LIN {X 0,Y 258.897,Z 434.556,A -85,B 0,C 180,E1 -20301.928,E2 -20301.928} C_VEL
LIN {X 0,Y 259.548,Z 434.776,A -85,B 0,C 180,E1 -20304.325,E2 -20304.325} C_VEL
LIN {X 0,Y 259.942,Z 436.236,A -85,B 0,C 180,E1 -20306.945,E2 -20306.945} C_VEL
LIN {X 0,Y 259.701,Z 437.624,A -85,B 0,C 180,E1 -20308.285,E2 -20308.285} C_VEL
LIN {X 0,Y 258.705,Z 439.082,A -85,B 0,C 180,E1 -20308.925,E2 -20308.925} C_VEL
LIN {X 0,Y 251.709,Z 446.598,A -85,B 0,C 180,E1 -20311.662,E2 -20311.662} C_VEL
LIN {X 0,Y 246.851,Z 451.078,A -85,B 0,C 180,E1 -20313.813,E2 -20313.813} C_VEL
LIN {X 0,Y 242.381,Z 454.631,A -85,B 0,C 180,E1 -20316.05,E2 -20316.05} C_VEL
LIN {X 0,Y 237.058,Z 458.044,A -85,B 0,C 180,E1 -20319.16,E2 -20319.16} C_VEL
LIN {X 0,Y 232.484,Z 459.981,A -85,B 0,C 180,E1 -20322.404,E2 -20322.404} C_VEL
LIN {X 0,Y 228.635,Z 460.543,A -85,B 0,C 180,E1 -20325.764,E2 -20325.764} C_VEL
LIN {X 0,Y 225.606,Z 459.628,A -85,B 0,C 180,E1 -20329.227,E2 -20329.227} C_VEL
LIN {X 0,Y 223.289,Z 457.297,A -85,B 0,C 180,E1 -20332.767,E2 -20332.767} C_VEL
LIN {X 0,Y 221.729,Z 453.432,A -85,B 0,C 180,E1 -20336.365,E2 -20336.365} C_VEL
LIN {X 0,Y 220.972,Z 447.998,A -85,B 0,C 180,E1 -20340,E2 -20340} C_VEL
LIN {X 0,Y 220.653,Z 441.734,A -85,B 0,C 180,E1 -20343.195,E2 -20343.195} C_VEL
LIN {X 0,Y 220.902,Z 433.929,A -85,B 0,C 180,E1 -20346.393,E2 -20346.393} C_VEL
LIN {X 0,Y 221.552,Z 425.762,A -85,B 0,C 180,E1 -20349.129,E2 -20349.129} C_VEL
LIN {X 0,Y 222.379,Z 415.886,A -85,B 0,C 180,E1 -20351.853,E2 -20351.853} C_VEL
LIN {X 0,Y 223.293,Z 404.919,A -85,B 0,C 180,E1 -20354.351,E2 -20354.351} C_VEL
LIN {X 0,Y 224.497,Z 392.799,A -85,B 0,C 180,E1 -20356.598,E2 -20356.598} C_VEL
LIN {X 0,Y 224.918,Z 385.6,A -85,B 0,C 180,E1 -20357.737,E2 -20357.737} C_VEL
LIN {X 0,Y 221.874,Z 372.126,A -85,B 0,C 180,E1 -20359.633,E2 -20359.633} C_VEL
LIN {X 0,Y 221.004,Z 367.954,A -85,B 0,C 180,E1 -20360.148,E2 -20360.148} C_VEL
LIN {X 0,Y 220.87,Z 367.97,A -85,B 0,C 180,E1 -20364.434,E2 -20364.434} C_VEL
LIN {X 0,Y 220.839,Z 367.975,A -85,B 0,C 180,E1 -20368.513,E2 -20368.513} C_VEL
LIN {X 0,Y 220.826,Z 367.978,A -85,B 0,C 180,E1 -20372.754,E2 -20372.754} C_VEL
LIN {X 0,Y 220.839,Z 367.976,A -85,B 0,C 180,E1 -20377.288,E2 -20377.288} C_VEL
LIN {X 0,Y 220.839,Z 367.975,A -85,B 0,C 180,E1 -20380.201,E2 -20380.201} C_VEL
LIN {X 0,Y 220.805,Z 367.978,A -85,B 0,C 180,E1 -20384.446,E2 -20384.446} C_VEL
LIN {X 0,Y 220.777,Z 367.983,A -85,B 0,C 180,E1 -20388.049,E2 -20388.049} C_VEL
LIN {X 0,Y 220.833,Z 367.977,A -85,B 0,C 180,E1 -20392.794,E2 -20392.794} C_VEL
LIN {X 0,Y 220.825,Z 367.976,A -85,B 0,C 180,E1 -20397.245,E2 -20397.245} C_VEL
LIN {X 0,Y 220.836,Z 367.973,A -85,B 0,C 180,E1 -20401.486,E2 -20401.486} C_VEL
LIN {X 0,Y 220.873,Z 367.97,A -85,B 0,C 180,E1 -20405.566,E2 -20405.566} C_VEL
LIN {X 0,Y 220.91,Z 367.963,A -85,B 0,C 180,E1 -20409.516,E2 -20409.516} C_VEL
LIN {X 0,Y 221.018,Z 367.952,A -85,B 0,C 180,E1 -20413.37,E2 -20413.37} C_VEL
LIN {X 0,Y 221.082,Z 367.943,A -85,B 0,C 180,E1 -20419.004,E2 -20419.004} C_VEL
LIN {X 0,Y 221.26,Z 367.922,A -85,B 0,C 180,E1 -20422.701,E2 -20422.701} C_VEL
LIN {X 0,Y 221.513,Z 367.893,A -85,B 0,C 180,E1 -20428.182,E2 -20428.182} C_VEL
LIN {X 0,Y 221.514,Z 367.893,A -85,B 0,C 180,E1 -20431.818,E2 -20431.818} C_VEL
LIN {X 0,Y 221.26,Z 367.922,A -85,B 0,C 180,E1 -20437.3,E2 -20437.3} C_VEL
LIN {X 0,Y 221.082,Z 367.943,A -85,B 0,C 180,E1 -20440.996,E2 -20440.996} C_VEL
LIN {X 0,Y 221.018,Z 367.952,A -85,B 0,C 180,E1 -20446.63,E2 -20446.63} C_VEL
LIN {X 0,Y 220.894,Z 367.965,A -85,B 0,C 180,E1 -20450.486,E2 -20450.486} C_VEL
LIN {X 0,Y 220.869,Z 367.971,A -85,B 0,C 180,E1 -20454.435,E2 -20454.435} C_VEL
LIN {X 0,Y 220.837,Z 367.973,A -85,B 0,C 180,E1 -20458.514,E2 -20458.514} C_VEL
LIN {X 0,Y 220.826,Z 367.976,A -85,B 0,C 180,E1 -20462.755,E2 -20462.755} C_VEL
LIN {X 0,Y 220.839,Z 367.976,A -85,B 0,C 180,E1 -20467.288,E2 -20467.288} C_VEL
LIN {X 0,Y 220.862,Z 367.972,A -85,B 0,C 180,E1 -20471.932,E2 -20471.932} C_VEL
LIN {X 0,Y 220.792,Z 367.98,A -85,B 0,C 180,E1 -20475.551,E2 -20475.551} C_VEL
LIN {X 0,Y 220.811,Z 367.978,A -85,B 0,C 180,E1 -20480.464,E2 -20480.464} C_VEL
LIN {X 0,Y 220.802,Z 367.979,A -85,B 0,C 180,E1 -20485.046,E2 -20485.046} C_VEL
LIN {X 0,Y 220.87,Z 367.972,A -85,B 0,C 180,E1 -20489.395,E2 -20489.395} C_VEL
LIN {X 0,Y 220.898,Z 367.964,A -85,B 0,C 180,E1 -20493.55,E2 -20493.55} C_VEL
LIN {X 0,Y 220.881,Z 367.97,A -85,B 0,C 180,E1 -20497.554,E2 -20497.554} C_VEL
LIN {X 0,Y 220.988,Z 367.956,A -85,B 0,C 180,E1 -20502.571,E2 -20502.571} C_VEL
LIN {X 0,Y 221.03,Z 367.952,A -85,B 0,C 180,E1 -20507.14,E2 -20507.14} C_VEL
LIN {X 0,Y 221.262,Z 367.921,A -85,B 0,C 180,E1 -20510.862,E2 -20510.862} C_VEL
LIN {X 0,Y 221.315,Z 367.916,A -85,B 0,C 180,E1 -20512.703,E2 -20512.703} C_VEL
LIN {X 0,Y 221.516,Z 367.891,A -85,B 0,C 180,E1 -20518.182,E2 -20518.182} C_VEL
LIN {X 0,Y 221.517,Z 367.889,A -85,B 0,C 180,E1 -20521.818,E2 -20521.818} C_VEL
LIN {X 0,Y 221.258,Z 367.92,A -85,B 0,C 180,E1 -20527.3,E2 -20527.3} C_VEL
LIN {X 0,Y 221.071,Z 367.945,A -85,B 0,C 180,E1 -20530.997,E2 -20530.997} C_VEL
LIN {X 0,Y 221,Z 367.954,A -85,B 0,C 180,E1 -20534.739,E2 -20534.739} C_VEL
LIN {X 0,Y 220.926,Z 367.964,A -85,B 0,C 180,E1 -20538.549,E2 -20538.549} C_VEL
LIN {X 0,Y 220.9,Z 367.967,A -85,B 0,C 180,E1 -20542.683,E2 -20542.683} C_VEL
LIN {X 0,Y 220.887,Z 367.967,A -85,B 0,C 180,E1 -20547.015,E2 -20547.015} C_VEL
LIN {X 0,Y 220.842,Z 367.974,A -85,B 0,C 180,E1 -20550.768,E2 -20550.768} C_VEL
LIN {X 0,Y 220.819,Z 367.974,A -85,B 0,C 180,E1 -20554.952,E2 -20554.952} C_VEL
LIN {X 0,Y 220.984,Z 367.957,A -85,B 0,C 180,E1 -20560.245,E2 -20560.245} C_VEL
LIN {X 0,Y 221.039,Z 368.08,A -85,B 0,C 180,E1 -20560.747,E2 -20560.747} C_VEL
LIN {X 0,Y 222.749,Z 377.209,A -85,B 0,C 180,E1 -20566.526,E2 -20566.526} C_VEL
LIN {X 0,Y 224.08,Z 383.095,A -85,B 0,C 180,E1 -20570.105,E2 -20570.105} C_VEL
LIN {X 0,Y 224.397,Z 385.506,A -85,B 0,C 180,E1 -20571.536,E2 -20571.536} C_VEL
LIN {X 0,Y 223.054,Z 392.251,A -85,B 0,C 180,E1 -20575.448,E2 -20575.448} C_VEL
LIN {X 0,Y 221.469,Z 400.97,A -85,B 0,C 180,E1 -20580.536,E2 -20580.536} C_VEL
LIN {X 0,Y 220.325,Z 410.683,A -85,B 0,C 180,E1 -20586.252,E2 -20586.252} C_VEL
LIN {X 0,Y 220.299,Z 410.997,A -85,B 0,C 180,E1 -20586.436,E2 -20586.436} C_VEL
LIN {X 0,Y 220.113,Z 423.689,A -85,B 0,C 180,E1 -20587.471,E2 -20587.471} C_VEL
LIN {X 0,Y 220.463,Z 437.057,A -85,B 0,C 180,E1 -20588.911,E2 -20588.911} C_VEL
LIN {X 0,Y 220.132,Z 442.349,A -85,B 0,C 180,E1 -20589.594,E2 -20589.594} C_VEL
LIN {X 0,Y 217.709,Z 450.666,A -85,B 0,C 180,E1 -20590.871,E2 -20590.871} C_VEL
LIN {X 0,Y 215.3,Z 458.611,A -85,B 0,C 180,E1 -20592.332,E2 -20592.332} C_VEL
LIN {X 0,Y 214.992,Z 463.305,A -85,B 0,C 180,E1 -20593.279,E2 -20593.279} C_VEL
LIN {X 0,Y 215.345,Z 468.453,A -85,B 0,C 180,E1 -20594.38,E2 -20594.38} C_VEL
LIN {X 0,Y 214.674,Z 477.726,A -85,B 0,C 180,E1 -20596.752,E2 -20596.752} C_VEL
LIN {X 0,Y 214.373,Z 486.701,A -85,B 0,C 180,E1 -20599.585,E2 -20599.585} C_VEL
LIN {X 0,Y 214.461,Z 494.06,A -85,B 0,C 180,E1 -20602.468,E2 -20602.468} C_VEL
LIN {X 0,Y 214.917,Z 499.835,A -85,B 0,C 180,E1 -20605.311,E2 -20605.311} C_VEL
LIN {X 0,Y 215.459,Z 504.208,A -85,B 0,C 180,E1 -20608.131,E2 -20608.131} C_VEL
LIN {X 0,Y 215.668,Z 506.362,A -85,B 0,C 180,E1 -20610,E2 -20610} C_VEL
LIN {X 0,Y 214.924,Z 507.775,A -85,B 0,C 180,E1 -20611.874,E2 -20611.874} C_VEL
LIN {X 0,Y 214.162,Z 508.735,A -85,B 0,C 180,E1 -20613.763,E2 -20613.763} C_VEL
LIN {X 0,Y 213.01,Z 509.516,A -85,B 0,C 180,E1 -20617.584,E2 -20617.584} C_VEL
LIN {X 0,Y 212.759,Z 508.905,A -85,B 0,C 180,E1 -20621.431,E2 -20621.431} C_VEL
LIN {X 0,Y 213.664,Z 507.003,A -85,B 0,C 180,E1 -20625.257,E2 -20625.257} C_VEL
LIN {X 0,Y 215.992,Z 503.521,A -85,B 0,C 180,E1 -20629.332,E2 -20629.332} C_VEL
LIN {X 0,Y 219.285,Z 499.472,A -85,B 0,C 180,E1 -20632.619,E2 -20632.619} C_VEL
LIN {X 0,Y 224.027,Z 493.791,A -85,B 0,C 180,E1 -20636.053,E2 -20636.053} C_VEL
LIN {X 0,Y 229.224,Z 486.787,A -85,B 0,C 180,E1 -20639.377,E2 -20639.377} C_VEL
LIN {X 0,Y 235.31,Z 478.403,A -85,B 0,C 180,E1 -20642.521,E2 -20642.521} C_VEL
LIN {X 0,Y 240.065,Z 470.429,A -85,B 0,C 180,E1 -20645.272,E2 -20645.272} C_VEL
LIN {X 0,Y 244.073,Z 462.536,A -85,B 0,C 180,E1 -20647.96,E2 -20647.96} C_VEL
LIN {X 0,Y 247.623,Z 454.754,A -85,B 0,C 180,E1 -20650.752,E2 -20650.752} C_VEL
LIN {X 0,Y 251.169,Z 447.148,A -85,B 0,C 180,E1 -20653.712,E2 -20653.712} C_VEL
LIN {X 0,Y 252.237,Z 444.781,A -85,B 0,C 180,E1 -20654.827,E2 -20654.827} C_VEL
LIN {X 0,Y 252.529,Z 443.033,A -85,B 0,C 180,E1 -20656.352,E2 -20656.352} C_VEL
LIN {X 0,Y 253.037,Z 441.118,A -85,B 0,C 180,E1 -20658.583,E2 -20658.583} C_VEL
LIN {X 0,Y 253.639,Z 439.942,A -85,B 0,C 180,E1 -20660.882,E2 -20660.882} C_VEL
LIN {X 0,Y 254.229,Z 439.583,A -85,B 0,C 180,E1 -20663.292,E2 -20663.292} C_VEL
LIN {X 0,Y 254.488,Z 439.791,A -85,B 0,C 180,E1 -20664.553,E2 -20664.553} C_VEL
LIN {X 0,Y 254.572,Z 440.686,A -85,B 0,C 180,E1 -20666.485,E2 -20666.485} C_VEL
LIN {X 0,Y 254.481,Z 441.386,A -85,B 0,C 180,E1 -20667.416,E2 -20667.416} C_VEL
LIN {X 0,Y 253.296,Z 442.857,A -85,B 0,C 180,E1 -20668.185,E2 -20668.185} C_VEL
LIN {X 0,Y 246.033,Z 449.795,A -85,B 0,C 180,E1 -20670.947,E2 -20670.947} C_VEL
LIN {X 0,Y 239.373,Z 455.094,A -85,B 0,C 180,E1 -20673.87,E2 -20673.87} C_VEL
LIN {X 0,Y 233.444,Z 458.797,A -85,B 0,C 180,E1 -20676.96,E2 -20676.96} C_VEL
LIN {X 0,Y 228.259,Z 461.111,A -85,B 0,C 180,E1 -20680.203,E2 -20680.203} C_VEL
LIN {X 0,Y 223.761,Z 462.001,A -85,B 0,C 180,E1 -20683.58,E2 -20683.58} C_VEL
LIN {X 0,Y 220.21,Z 461.481,A -85,B 0,C 180,E1 -20687.091,E2 -20687.091} C_VEL
LIN {X 0,Y 217.379,Z 459.554,A -85,B 0,C 180,E1 -20690.697,E2 -20690.697} C_VEL
LIN {X 0,Y 215.348,Z 456.131,A -85,B 0,C 180,E1 -20694.381,E2 -20694.381} C_VEL
LIN {X 0,Y 214.194,Z 451.191,A -85,B 0,C 180,E1 -20698.119,E2 -20698.119} C_VEL
LIN {X 0,Y 213.749,Z 446.372,A -85,B 0,C 180,E1 -20700.942,E2 -20700.942} C_VEL
LIN {X 0,Y 213.555,Z 439.379,A -85,B 0,C 180,E1 -20704.246,E2 -20704.246} C_VEL
LIN {X 0,Y 214.061,Z 430.752,A -85,B 0,C 180,E1 -20707.546,E2 -20707.546} C_VEL
LIN {X 0,Y 214.668,Z 422.303,A -85,B 0,C 180,E1 -20710.194,E2 -20710.194} C_VEL
LIN {X 0,Y 215.588,Z 412.708,A -85,B 0,C 180,E1 -20712.711,E2 -20712.711} C_VEL
LIN {X 0,Y 216.499,Z 402.058,A -85,B 0,C 180,E1 -20715.052,E2 -20715.052} C_VEL
LIN {X 0,Y 217.767,Z 389.029,A -85,B 0,C 180,E1 -20717.369,E2 -20717.369} C_VEL
LIN {X 0,Y 217.714,Z 385.924,A -85,B 0,C 180,E1 -20717.858,E2 -20717.858} C_VEL
LIN {X 0,Y 214.889,Z 373.38,A -85,B 0,C 180,E1 -20719.673,E2 -20719.673} C_VEL
LIN {X 0,Y 213.971,Z 368.83,A -85,B 0,C 180,E1 -20720.299,E2 -20720.299} C_VEL
LIN {X 0,Y 213.804,Z 368.85,A -85,B 0,C 180,E1 -20725.298,E2 -20725.298} C_VEL
LIN {X 0,Y 213.782,Z 368.854,A -85,B 0,C 180,E1 -20729.545,E2 -20729.545} C_VEL
LIN {X 0,Y 213.771,Z 368.852,A -85,B 0,C 180,E1 -20733.979,E2 -20733.979} C_VEL
LIN {X 0,Y 213.78,Z 368.856,A -85,B 0,C 180,E1 -20738.654,E2 -20738.654} C_VEL
LIN {X 0,Y 213.776,Z 368.852,A -85,B 0,C 180,E1 -20743.675,E2 -20743.675} C_VEL
LIN {X 0,Y 213.718,Z 368.863,A -85,B 0,C 180,E1 -20748.876,E2 -20748.876} C_VEL
LIN {X 0,Y 213.754,Z 368.856,A -85,B 0,C 180,E1 -20753.713,E2 -20753.713} C_VEL
LIN {X 0,Y 213.796,Z 368.851,A -85,B 0,C 180,E1 -20758.724,E2 -20758.724} C_VEL
LIN {X 0,Y 213.826,Z 368.851,A -85,B 0,C 180,E1 -20762.603,E2 -20762.603} C_VEL
LIN {X 0,Y 213.863,Z 368.842,A -85,B 0,C 180,E1 -20766.946,E2 -20766.946} C_VEL
LIN {X 0,Y 213.934,Z 368.838,A -85,B 0,C 180,E1 -20772.304,E2 -20772.304} C_VEL
LIN {X 0,Y 213.954,Z 368.829,A -85,B 0,C 180,E1 -20776.707,E2 -20776.707} C_VEL
LIN {X 0,Y 214.143,Z 368.81,A -85,B 0,C 180,E1 -20780.555,E2 -20780.555} C_VEL
LIN {X 0,Y 214.102,Z 368.813,A -85,B 0,C 180,E1 -20784.349,E2 -20784.349} C_VEL
LIN {X 0,Y 214.447,Z 368.774,A -85,B 0,C 180,E1 -20788.122,E2 -20788.122} C_VEL
LIN {X 0,Y 214.551,Z 368.761,A -85,B 0,C 180,E1 -20790,E2 -20790} C_VEL
LIN {X 0,Y 214.447,Z 368.773,A -85,B 0,C 180,E1 -20791.878,E2 -20791.878} C_VEL
LIN {X 0,Y 214.2,Z 368.803,A -85,B 0,C 180,E1 -20797.542,E2 -20797.542} C_VEL
LIN {X 0,Y 214.009,Z 368.825,A -85,B 0,C 180,E1 -20801.364,E2 -20801.364} C_VEL
LIN {X 0,Y 213.935,Z 368.834,A -85,B 0,C 180,E1 -20805.237,E2 -20805.237} C_VEL
LIN {X 0,Y 213.87,Z 368.843,A -85,B 0,C 180,E1 -20809.185,E2 -20809.185} C_VEL
LIN {X 0,Y 213.848,Z 368.845,A -85,B 0,C 180,E1 -20813.227,E2 -20813.227} C_VEL
LIN {X 0,Y 213.83,Z 368.851,A -85,B 0,C 180,E1 -20817.45,E2 -20817.45} C_VEL
LIN {X 0,Y 213.781,Z 368.855,A -85,B 0,C 180,E1 -20821.736,E2 -20821.736} C_VEL
LIN {X 0,Y 213.756,Z 368.856,A -85,B 0,C 180,E1 -20826.286,E2 -20826.286} C_VEL
LIN {X 0,Y 213.799,Z 368.853,A -85,B 0,C 180,E1 -20831.106,E2 -20831.106} C_VEL
LIN {X 0,Y 213.81,Z 368.851,A -85,B 0,C 180,E1 -20833.685,E2 -20833.685} C_VEL
LIN {X 0,Y 213.749,Z 368.855,A -85,B 0,C 180,E1 -20836.333,E2 -20836.333} C_VEL
LIN {X 0,Y 213.727,Z 368.863,A -85,B 0,C 180,E1 -20841.334,E2 -20841.334} C_VEL
LIN {X 0,Y 213.758,Z 368.853,A -85,B 0,C 180,E1 -20846.018,E2 -20846.018} C_VEL
LIN {X 0,Y 213.783,Z 368.854,A -85,B 0,C 180,E1 -20850.455,E2 -20850.455} C_VEL
LIN {X 0,Y 213.805,Z 368.849,A -85,B 0,C 180,E1 -20854.702,E2 -20854.702} C_VEL
LIN {X 0,Y 213.817,Z 368.853,A -85,B 0,C 180,E1 -20858.804,E2 -20858.804} C_VEL
LIN {X 0,Y 213.947,Z 368.833,A -85,B 0,C 180,E1 -20862.804,E2 -20862.804} C_VEL
LIN {X 0,Y 213.985,Z 368.832,A -85,B 0,C 180,E1 -20866.709,E2 -20866.709} C_VEL
LIN {X 0,Y 214.2,Z 368.802,A -85,B 0,C 180,E1 -20870.558,E2 -20870.558} C_VEL
LIN {X 0,Y 214.252,Z 368.794,A -85,B 0,C 180,E1 -20872.461,E2 -20872.461} C_VEL
LIN {X 0,Y 214.45,Z 368.771,A -85,B 0,C 180,E1 -20878.122,E2 -20878.122} C_VEL
LIN {X 0,Y 214.554,Z 368.755,A -85,B 0,C 180,E1 -20880,E2 -20880} C_VEL
LIN {X 0,Y 214.45,Z 368.769,A -85,B 0,C 180,E1 -20881.878,E2 -20881.878} C_VEL
LIN {X 0,Y 214.198,Z 368.8,A -85,B 0,C 180,E1 -20887.542,E2 -20887.542} C_VEL
LIN {X 0,Y 214.003,Z 368.826,A -85,B 0,C 180,E1 -20891.364,E2 -20891.364} C_VEL
LIN {X 0,Y 213.938,Z 368.833,A -85,B 0,C 180,E1 -20895.237,E2 -20895.237} C_VEL
LIN {X 0,Y 213.844,Z 368.845,A -85,B 0,C 180,E1 -20899.187,E2 -20899.187} C_VEL
LIN {X 0,Y 213.851,Z 368.844,A -85,B 0,C 180,E1 -20903.227,E2 -20903.227} C_VEL
LIN {X 0,Y 213.832,Z 368.846,A -85,B 0,C 180,E1 -20907.45,E2 -20907.45} C_VEL
LIN {X 0,Y 213.773,Z 368.857,A -85,B 0,C 180,E1 -20911.737,E2 -20911.737} C_VEL
LIN {X 0,Y 213.76,Z 368.857,A -85,B 0,C 180,E1 -20916.285,E2 -20916.285} C_VEL
LIN {X 0,Y 213.979,Z 368.888,A -85,B 0,C 180,E1 -20920.687,E2 -20920.687} C_VEL
LIN {X 0,Y 215.44,Z 376.781,A -85,B 0,C 180,E1 -20925.863,E2 -20925.863} C_VEL
LIN {X 0,Y 217.06,Z 383.878,A -85,B 0,C 180,E1 -20930.343,E2 -20930.343} C_VEL
LIN {X 0,Y 217.147,Z 386.687,A -85,B 0,C 180,E1 -20932.052,E2 -20932.052} C_VEL
LIN {X 0,Y 215.652,Z 393.822,A -85,B 0,C 180,E1 -20936.356,E2 -20936.356} C_VEL
LIN {X 0,Y 213.908,Z 404.111,A -85,B 0,C 180,E1 -20942.614,E2 -20942.614} C_VEL
LIN {X 0,Y 213.252,Z 410.025,A -85,B 0,C 180,E1 -20946.254,E2 -20946.254} C_VEL
LIN {X 0,Y 213.031,Z 424.1,A -85,B 0,C 180,E1 -20947.48,E2 -20947.48} C_VEL
LIN {X 0,Y 213.397,Z 437.408,A -85,B 0,C 180,E1 -20949.013,E2 -20949.013} C_VEL
LIN {X 0,Y 214.013,Z 449.844,A -85,B 0,C 180,E1 -20950.829,E2 -20950.829} C_VEL
LIN {X 0,Y 214.824,Z 461.312,A -85,B 0,C 180,E1 -20952.876,E2 -20952.876} C_VEL
LIN {X 0,Y 214.992,Z 463.305,A -85,B 0,C 180,E1 -20953.279,E2 -20953.279} C_VEL
LIN {X 0,Y 214.865,Z 466.366,A -85,B 0,C 180,E1 -20953.935,E2 -20953.935} C_VEL
LIN {X 0,Y 213.575,Z 470.619,A -85,B 0,C 180,E1 -20954.981,E2 -20954.981} C_VEL
LIN {X 0,Y 208.863,Z 479.328,A -85,B 0,C 180,E1 -20957.684,E2 -20957.684} C_VEL
LIN {X 0,Y 207.618,Z 482.941,A -85,B 0,C 180,E1 -20958.966,E2 -20958.966} C_VEL
LIN {X 0,Y 207.486,Z 484.164,A -85,B 0,C 180,E1 -20959.405,E2 -20959.405} C_VEL
LIN {X 0,Y 207.583,Z 491.366,A -85,B 0,C 180,E1 -20962.217,E2 -20962.217} C_VEL
LIN {X 0,Y 207.989,Z 497.394,A -85,B 0,C 180,E1 -20965.154,E2 -20965.154} C_VEL
LIN {X 0,Y 208.583,Z 502.045,A -85,B 0,C 180,E1 -20968.069,E2 -20968.069} C_VEL
LIN {X 0,Y 208.814,Z 504.383,A -85,B 0,C 180,E1 -20970,E2 -20970} C_VEL
LIN {X 0,Y 208.039,Z 505.905,A -85,B 0,C 180,E1 -20971.936,E2 -20971.936} C_VEL
LIN {X 0,Y 207.238,Z 506.957,A -85,B 0,C 180,E1 -20973.889,E2 -20973.889} C_VEL
LIN {X 0,Y 206.006,Z 507.927,A -85,B 0,C 180,E1 -20977.843,E2 -20977.843} C_VEL
LIN {X 0,Y 205.809,Z 507.58,A -85,B 0,C 180,E1 -20981.823,E2 -20981.823} C_VEL
LIN {X 0,Y 206.79,Z 505.98,A -85,B 0,C 180,E1 -20985.777,E2 -20985.777} C_VEL
LIN {X 0,Y 209.079,Z 503.076,A -85,B 0,C 180,E1 -20989.745,E2 -20989.745} C_VEL
LIN {X 0,Y 212.729,Z 499.155,A -85,B 0,C 180,E1 -20993.356,E2 -20993.356} C_VEL
LIN {X 0,Y 217.652,Z 493.871,A -85,B 0,C 180,E1 -20996.876,E2 -20996.876} C_VEL
LIN {X 0,Y 223.08,Z 487.324,A -85,B 0,C 180,E1 -21000.27,E2 -21000.27} C_VEL
LIN {X 0,Y 229.425,Z 479.514,A -85,B 0,C 180,E1 -21003.463,E2 -21003.463} C_VEL
LIN {X 0,Y 234.288,Z 472.337,A -85,B 0,C 180,E1 -21006.146,E2 -21006.146} C_VEL
LIN {X 0,Y 238.941,Z 464.382,A -85,B 0,C 180,E1 -21009.084,E2 -21009.084} C_VEL
LIN {X 0,Y 244.322,Z 454.352,A -85,B 0,C 180,E1 -21013.021,E2 -21013.021} C_VEL
LIN {X 0,Y 247.112,Z 449.26,A -85,B 0,C 180,E1 -21015.318,E2 -21015.318} C_VEL
LIN {X 0,Y 247.615,Z 446.997,A -85,B 0,C 180,E1 -21017.558,E2 -21017.558} C_VEL
LIN {X 0,Y 248.211,Z 445.381,A -85,B 0,C 180,E1 -21019.862,E2 -21019.862} C_VEL
LIN {X 0,Y 248.776,Z 444.499,A -85,B 0,C 180,E1 -21022.28,E2 -21022.28} C_VEL
LIN {X 0,Y 249.049,Z 444.399,A -85,B 0,C 180,E1 -21023.657,E2 -21023.657} C_VEL
LIN {X 0,Y 249.121,Z 444.877,A -85,B 0,C 180,E1 -21025.651,E2 -21025.651} C_VEL
LIN {X 0,Y 247.957,Z 446.555,A -85,B 0,C 180,E1 -21027.416,E2 -21027.416} C_VEL
LIN {X 0,Y 240.401,Z 452.958,A -85,B 0,C 180,E1 -21030.199,E2 -21030.199} C_VEL
LIN {X 0,Y 233.444,Z 457.739,A -85,B 0,C 180,E1 -21033.154,E2 -21033.154} C_VEL
LIN {X 0,Y 227.276,Z 461.062,A -85,B 0,C 180,E1 -21036.297,E2 -21036.297} C_VEL
LIN {X 0,Y 221.819,Z 462.953,A -85,B 0,C 180,E1 -21039.603,E2 -21039.603} C_VEL
LIN {X 0,Y 217.117,Z 463.514,A -85,B 0,C 180,E1 -21043.062,E2 -21043.062} C_VEL
LIN {X 0,Y 213.407,Z 462.634,A -85,B 0,C 180,E1 -21046.672,E2 -21046.672} C_VEL
LIN {X 0,Y 210.445,Z 460.353,A -85,B 0,C 180,E1 -21050.387,E2 -21050.387} C_VEL
LIN {X 0,Y 208.302,Z 456.64,A -85,B 0,C 180,E1 -21054.19,E2 -21054.19} C_VEL
LIN {X 0,Y 207.102,Z 451.338,A -85,B 0,C 180,E1 -21058.055,E2 -21058.055} C_VEL
LIN {X 0,Y 206.655,Z 446.258,A -85,B 0,C 180,E1 -21060.974,E2 -21060.974} C_VEL
LIN {X 0,Y 206.487,Z 438.984,A -85,B 0,C 180,E1 -21064.392,E2 -21064.392} C_VEL
LIN {X 0,Y 207.028,Z 429.957,A -85,B 0,C 180,E1 -21067.804,E2 -21067.804} C_VEL
LIN {X 0,Y 207.609,Z 421.66,A -85,B 0,C 180,E1 -21070.401,E2 -21070.401} C_VEL
LIN {X 0,Y 208.63,Z 411.198,A -85,B 0,C 180,E1 -21073.143,E2 -21073.143} C_VEL
LIN {X 0,Y 209.74,Z 398.784,A -85,B 0,C 180,E1 -21075.798,E2 -21075.798} C_VEL
LIN {X 0,Y 210.745,Z 388.038,A -85,B 0,C 180,E1 -21077.681,E2 -21077.681} C_VEL
LIN {X 0,Y 208.156,Z 375.772,A -85,B 0,C 180,E1 -21079.534,E2 -21079.534} C_VEL
LIN {X 0,Y 206.939,Z 369.706,A -85,B 0,C 180,E1 -21080.371,E2 -21080.371} C_VEL
LIN {X 0,Y 206.766,Z 369.726,A -85,B 0,C 180,E1 -21084.072,E2 -21084.072} C_VEL
LIN {X 0,Y 206.746,Z 369.73,A -85,B 0,C 180,E1 -21088.418,E2 -21088.418} C_VEL
LIN {X 0,Y 206.711,Z 369.735,A -85,B 0,C 180,E1 -21092.955,E2 -21092.955} C_VEL
LIN {X 0,Y 206.725,Z 369.733,A -85,B 0,C 180,E1 -21097.73,E2 -21097.73} C_VEL
LIN {X 0,Y 206.694,Z 369.734,A -85,B 0,C 180,E1 -21101.579,E2 -21101.579} C_VEL
LIN {X 0,Y 206.639,Z 369.743,A -85,B 0,C 180,E1 -21105.58,E2 -21105.58} C_VEL
LIN {X 0,Y 206.668,Z 369.738,A -85,B 0,C 180,E1 -21109.75,E2 -21109.75} C_VEL
LIN {X 0,Y 206.732,Z 369.735,A -85,B 0,C 180,E1 -21114.695,E2 -21114.695} C_VEL
LIN {X 0,Y 206.724,Z 369.73,A -85,B 0,C 180,E1 -21119.339,E2 -21119.339} C_VEL
LIN {X 0,Y 206.735,Z 369.732,A -85,B 0,C 180,E1 -21123.772,E2 -21123.772} C_VEL
LIN {X 0,Y 206.779,Z 369.725,A -85,B 0,C 180,E1 -21128.046,E2 -21128.046} C_VEL
LIN {X 0,Y 206.879,Z 369.716,A -85,B 0,C 180,E1 -21132.197,E2 -21132.197} C_VEL
LIN {X 0,Y 206.896,Z 369.711,A -85,B 0,C 180,E1 -21136.244,E2 -21136.244} C_VEL
LIN {X 0,Y 207.1,Z 369.689,A -85,B 0,C 180,E1 -21140.231,E2 -21140.231} C_VEL
LIN {X 0,Y 207.063,Z 369.691,A -85,B 0,C 180,E1 -21144.156,E2 -21144.156} C_VEL
LIN {X 0,Y 207.383,Z 369.653,A -85,B 0,C 180,E1 -21148.058,E2 -21148.058} C_VEL
LIN {X 0,Y 207.516,Z 369.638,A -85,B 0,C 180,E1 -21150,E2 -21150} C_VEL
LIN {X 0,Y 207.384,Z 369.653,A -85,B 0,C 180,E1 -21151.942,E2 -21151.942} C_VEL
LIN {X 0,Y 207.142,Z 369.683,A -85,B 0,C 180,E1 -21157.8,E2 -21157.8} C_VEL
LIN {X 0,Y 206.932,Z 369.707,A -85,B 0,C 180,E1 -21161.758,E2 -21161.758} C_VEL
LIN {X 0,Y 206.869,Z 369.718,A -85,B 0,C 180,E1 -21165.771,E2 -21165.771} C_VEL
LIN {X 0,Y 206.801,Z 369.723,A -85,B 0,C 180,E1 -21169.868,E2 -21169.868} C_VEL
LIN {X 0,Y 206.765,Z 369.729,A -85,B 0,C 180,E1 -21174.072,E2 -21174.072} C_VEL
LIN {X 0,Y 206.745,Z 369.728,A -85,B 0,C 180,E1 -21178.419,E2 -21178.419} C_VEL
LIN {X 0,Y 206.711,Z 369.735,A -85,B 0,C 180,E1 -21182.956,E2 -21182.956} C_VEL
LIN {X 0,Y 206.727,Z 369.73,A -85,B 0,C 180,E1 -21187.73,E2 -21187.73} C_VEL
LIN {X 0,Y 206.727,Z 369.734,A -85,B 0,C 180,E1 -21191.59,E2 -21191.59} C_VEL
LIN {X 0,Y 206.676,Z 369.738,A -85,B 0,C 180,E1 -21195.57,E2 -21195.57} C_VEL
LIN {X 0,Y 206.669,Z 369.74,A -85,B 0,C 180,E1 -21199.751,E2 -21199.751} C_VEL
LIN {X 0,Y 206.701,Z 369.735,A -85,B 0,C 180,E1 -21204.689,E2 -21204.689} C_VEL
LIN {X 0,Y 206.726,Z 369.734,A -85,B 0,C 180,E1 -21209.34,E2 -21209.34} C_VEL
LIN {X 0,Y 206.735,Z 369.728,A -85,B 0,C 180,E1 -21213.773,E2 -21213.773} C_VEL
LIN {X 0,Y 206.761,Z 369.728,A -85,B 0,C 180,E1 -21218.044,E2 -21218.044} C_VEL
LIN {X 0,Y 206.88,Z 369.712,A -85,B 0,C 180,E1 -21222.197,E2 -21222.197} C_VEL
LIN {X 0,Y 206.918,Z 369.709,A -85,B 0,C 180,E1 -21226.246,E2 -21226.246} C_VEL
LIN {X 0,Y 207.137,Z 369.681,A -85,B 0,C 180,E1 -21230.233,E2 -21230.233} C_VEL
LIN {X 0,Y 207.193,Z 369.672,A -85,B 0,C 180,E1 -21232.202,E2 -21232.202} C_VEL
LIN {X 0,Y 207.386,Z 369.651,A -85,B 0,C 180,E1 -21238.058,E2 -21238.058} C_VEL
LIN {X 0,Y 207.519,Z 369.631,A -85,B 0,C 180,E1 -21240,E2 -21240} C_VEL
LIN {X 0,Y 207.386,Z 369.649,A -85,B 0,C 180,E1 -21241.942,E2 -21241.942} C_VEL
LIN {X 0,Y 207.141,Z 369.679,A -85,B 0,C 180,E1 -21247.8,E2 -21247.8} C_VEL
LIN {X 0,Y 206.929,Z 369.708,A -85,B 0,C 180,E1 -21251.758,E2 -21251.758} C_VEL
LIN {X 0,Y 206.872,Z 369.714,A -85,B 0,C 180,E1 -21255.771,E2 -21255.771} C_VEL
LIN {X 0,Y 206.788,Z 369.726,A -85,B 0,C 180,E1 -21259.869,E2 -21259.869} C_VEL
LIN {X 0,Y 206.767,Z 369.728,A -85,B 0,C 180,E1 -21264.072,E2 -21264.072} C_VEL
LIN {X 0,Y 206.74,Z 369.732,A -85,B 0,C 180,E1 -21268.42,E2 -21268.42} C_VEL
LIN {X 0,Y 206.709,Z 369.733,A -85,B 0,C 180,E1 -21272.956,E2 -21272.956} C_VEL
LIN {X 0,Y 206.737,Z 369.733,A -85,B 0,C 180,E1 -21277.728,E2 -21277.728} C_VEL
LIN {X 0,Y 206.942,Z 369.819,A -85,B 0,C 180,E1 -21280.755,E2 -21280.755} C_VEL
LIN {X 0,Y 208.56,Z 378.207,A -85,B 0,C 180,E1 -21286.428,E2 -21286.428} C_VEL
LIN {X 0,Y 210.007,Z 384.49,A -85,B 0,C 180,E1 -21290.517,E2 -21290.517} C_VEL
LIN {X 0,Y 210.076,Z 386.448,A -85,B 0,C 180,E1 -21291.763,E2 -21291.763} C_VEL
LIN {X 0,Y 208.593,Z 393.556,A -85,B 0,C 180,E1 -21296.225,E2 -21296.225} C_VEL
LIN {X 0,Y 206.766,Z 404.081,A -85,B 0,C 180,E1 -21302.885,E2 -21302.885} C_VEL
LIN {X 0,Y 206.235,Z 409.081,A -85,B 0,C 180,E1 -21306.099,E2 -21306.099} C_VEL
LIN {X 0,Y 205.912,Z 422.074,A -85,B 0,C 180,E1 -21307.261,E2 -21307.261} C_VEL
LIN {X 0,Y 206.213,Z 434.967,A -85,B 0,C 180,E1 -21308.77,E2 -21308.77} C_VEL
LIN {X 0,Y 206.871,Z 448.445,A -85,B 0,C 180,E1 -21310.786,E2 -21310.786} C_VEL
LIN {X 0,Y 207.761,Z 460.586,A -85,B 0,C 180,E1 -21313.036,E2 -21313.036} C_VEL
LIN {X 0,Y 208.324,Z 467.686,A -85,B 0,C 180,E1 -21314.593,E2 -21314.593} C_VEL
LIN {X 0,Y 207.679,Z 477.654,A -85,B 0,C 180,E1 -21317.293,E2 -21317.293} C_VEL
LIN {X 0,Y 207.486,Z 484.164,A -85,B 0,C 180,E1 -21319.405,E2 -21319.405} C_VEL
LIN {X 0,Y 206.795,Z 487.552,A -85,B 0,C 180,E1 -21320.733,E2 -21320.733} C_VEL
LIN {X 0,Y 204.234,Z 492.196,A -85,B 0,C 180,E1 -21323.066,E2 -21323.066} C_VEL
LIN {X 0,Y 202.229,Z 495.405,A -85,B 0,C 180,E1 -21325.055,E2 -21325.055} C_VEL
LIN {X 0,Y 201.523,Z 497.722,A -85,B 0,C 180,E1 -21326.605,E2 -21326.605} C_VEL
LIN {X 0,Y 201.539,Z 498.493,A -85,B 0,C 180,E1 -21327.126,E2 -21327.126} C_VEL
LIN {X 0,Y 201.988,Z 502.28,A -85,B 0,C 180,E1 -21330,E2 -21330} C_VEL
LIN {X 0,Y 201.198,Z 503.919,A -85,B 0,C 180,E1 -21332.002,E2 -21332.002} C_VEL
LIN {X 0,Y 200.34,Z 505.097,A -85,B 0,C 180,E1 -21334.023,E2 -21334.023} C_VEL
LIN {X 0,Y 199.046,Z 506.304,A -85,B 0,C 180,E1 -21338.119,E2 -21338.119} C_VEL
LIN {X 0,Y 198.875,Z 506.215,A -85,B 0,C 180,E1 -21342.241,E2 -21342.241} C_VEL
LIN {X 0,Y 199.938,Z 504.896,A -85,B 0,C 180,E1 -21346.332,E2 -21346.332} C_VEL
LIN {X 0,Y 202.315,Z 502.386,A -85,B 0,C 180,E1 -21350.327,E2 -21350.327} C_VEL
LIN {X 0,Y 206.222,Z 498.728,A -85,B 0,C 180,E1 -21354.139,E2 -21354.139} C_VEL
LIN {X 0,Y 211.333,Z 493.864,A -85,B 0,C 180,E1 -21357.748,E2 -21357.748} C_VEL
LIN {X 0,Y 216.988,Z 487.794,A -85,B 0,C 180,E1 -21361.213,E2 -21361.213} C_VEL
LIN {X 0,Y 223.593,Z 480.536,A -85,B 0,C 180,E1 -21364.456,E2 -21364.456} C_VEL
LIN {X 0,Y 228.75,Z 473.772,A -85,B 0,C 180,E1 -21367.202,E2 -21367.202} C_VEL
LIN {X 0,Y 233.824,Z 466.179,A -85,B 0,C 180,E1 -21370.252,E2 -21370.252} C_VEL
LIN {X 0,Y 238.943,Z 457.959,A -85,B 0,C 180,E1 -21373.726,E2 -21373.726} C_VEL
LIN {X 0,Y 241.662,Z 453.735,A -85,B 0,C 180,E1 -21375.735,E2 -21375.735} C_VEL
LIN {X 0,Y 242.409,Z 451.303,A -85,B 0,C 180,E1 -21378.177,E2 -21378.177} C_VEL
LIN {X 0,Y 243.14,Z 449.464,A -85,B 0,C 180,E1 -21381.301,E2 -21381.301} C_VEL
LIN {X 0,Y 243.602,Z 448.978,A -85,B 0,C 180,E1 -21383.883,E2 -21383.883} C_VEL
LIN {X 0,Y 243.62,Z 449.044,A -85,B 0,C 180,E1 -21384.762,E2 -21384.762} C_VEL
LIN {X 0,Y 242.629,Z 450.211,A -85,B 0,C 180,E1 -21386.608,E2 -21386.608} C_VEL
LIN {X 0,Y 234.792,Z 456.026,A -85,B 0,C 180,E1 -21389.412,E2 -21389.412} C_VEL
LIN {X 0,Y 231.064,Z 458.406,A -85,B 0,C 180,E1 -21390.879,E2 -21390.879} C_VEL
LIN {X 0,Y 224.202,Z 461.978,A -85,B 0,C 180,E1 -21393.969,E2 -21393.969} C_VEL
LIN {X 0,Y 218.151,Z 464.173,A -85,B 0,C 180,E1 -21397.257,E2 -21397.257} C_VEL
LIN {X 0,Y 212.855,Z 465.007,A -85,B 0,C 180,E1 -21400.72,E2 -21400.72} C_VEL
LIN {X 0,Y 208.427,Z 464.481,A -85,B 0,C 180,E1 -21404.35,E2 -21404.35} C_VEL
LIN {X 0,Y 204.939,Z 462.588,A -85,B 0,C 180,E1 -21408.126,E2 -21408.126} C_VEL
LIN {X 0,Y 202.297,Z 459.231,A -85,B 0,C 180,E1 -21412.012,E2 -21412.012} C_VEL
LIN {X 0,Y 200.503,Z 454.42,A -85,B 0,C 180,E1 -21415.98,E2 -21415.98} C_VEL
LIN {X 0,Y 199.9,Z 449.727,A -85,B 0,C 180,E1 -21418.992,E2 -21418.992} C_VEL
LIN {X 0,Y 199.413,Z 442.984,A -85,B 0,C 180,E1 -21422.525,E2 -21422.525} C_VEL
LIN {X 0,Y 199.53,Z 434.617,A -85,B 0,C 180,E1 -21426.065,E2 -21426.065} C_VEL
LIN {X 0,Y 200.281,Z 425.977,A -85,B 0,C 180,E1 -21429.085,E2 -21429.085} C_VEL
LIN {X 0,Y 201.111,Z 415.496,A -85,B 0,C 180,E1 -21432.103,E2 -21432.103} C_VEL
LIN {X 0,Y 202.147,Z 403.865,A -85,B 0,C 180,E1 -21434.857,E2 -21434.857} C_VEL
LIN {X 0,Y 203.454,Z 390.92,A -85,B 0,C 180,E1 -21437.333,E2 -21437.333} C_VEL
LIN {X 0,Y 203.595,Z 387.9,A -85,B 0,C 180,E1 -21437.84,E2 -21437.84} C_VEL
LIN {X 0,Y 200.896,Z 375.694,A -85,B 0,C 180,E1 -21439.72,E2 -21439.72} C_VEL
LIN {X 0,Y 199.879,Z 370.585,A -85,B 0,C 180,E1 -21440.443,E2 -21440.443} C_VEL
LIN {X 0,Y 199.675,Z 370.61,A -85,B 0,C 180,E1 -21444.984,E2 -21444.984} C_VEL
LIN {X 0,Y 199.676,Z 370.612,A -85,B 0,C 180,E1 -21449.522,E2 -21449.522} C_VEL
LIN {X 0,Y 199.666,Z 370.612,A -85,B 0,C 180,E1 -21452.352,E2 -21452.352} C_VEL
LIN {X 0,Y 199.654,Z 370.615,A -85,B 0,C 180,E1 -21456.756,E2 -21456.756} C_VEL
LIN {X 0,Y 199.676,Z 370.611,A -85,B 0,C 180,E1 -21459.312,E2 -21459.312} C_VEL
LIN {X 0,Y 199.63,Z 370.615,A -85,B 0,C 180,E1 -21462.327,E2 -21462.327} C_VEL
LIN {X 0,Y 199.598,Z 370.621,A -85,B 0,C 180,E1 -21465.233,E2 -21465.233} C_VEL
LIN {X 0,Y 199.642,Z 370.614,A -85,B 0,C 180,E1 -21470.756,E2 -21470.756} C_VEL
LIN {X 0,Y 199.635,Z 370.616,A -85,B 0,C 180,E1 -21475.718,E2 -21475.718} C_VEL
LIN {X 0,Y 199.705,Z 370.608,A -85,B 0,C 180,E1 -21478.138,E2 -21478.138} C_VEL
LIN {X 0,Y 199.688,Z 370.611,A -85,B 0,C 180,E1 -21482.772,E2 -21482.772} C_VEL
LIN {X 0,Y 199.751,Z 370.599,A -85,B 0,C 180,E1 -21487.231,E2 -21487.231} C_VEL
LIN {X 0,Y 199.838,Z 370.591,A -85,B 0,C 180,E1 -21491.722,E2 -21491.722} C_VEL
LIN {X 0,Y 199.837,Z 370.59,A -85,B 0,C 180,E1 -21495.748,E2 -21495.748} C_VEL
LIN {X 0,Y 200.023,Z 370.568,A -85,B 0,C 180,E1 -21499.882,E2 -21499.882} C_VEL
LIN {X 0,Y 200.025,Z 370.569,A -85,B 0,C 180,E1 -21503.949,E2 -21503.949} C_VEL
LIN {X 0,Y 200.323,Z 370.531,A -85,B 0,C 180,E1 -21507.99,E2 -21507.99} C_VEL
LIN {X 0,Y 200.48,Z 370.514,A -85,B 0,C 180,E1 -21510,E2 -21510} C_VEL
LIN {X 0,Y 200.031,Z 370.565,A -85,B 0,C 180,E1 -21514.03,E2 -21514.03} C_VEL
LIN {X 0,Y 200.09,Z 370.562,A -85,B 0,C 180,E1 -21518.077,E2 -21518.077} C_VEL
LIN {X 0,Y 199.88,Z 370.582,A -85,B 0,C 180,E1 -21522.179,E2 -21522.179} C_VEL
LIN {X 0,Y 199.807,Z 370.595,A -85,B 0,C 180,E1 -21526.344,E2 -21526.344} C_VEL
LIN {X 0,Y 199.825,Z 370.592,A -85,B 0,C 180,E1 -21528.454,E2 -21528.454} C_VEL
LIN {X 0,Y 199.738,Z 370.605,A -85,B 0,C 180,E1 -21533.818,E2 -21533.818} C_VEL
LIN {X 0,Y 199.713,Z 370.604,A -85,B 0,C 180,E1 -21538.387,E2 -21538.387} C_VEL
LIN {X 0,Y 199.665,Z 370.611,A -85,B 0,C 180,E1 -21542.353,E2 -21542.353} C_VEL
LIN {X 0,Y 199.655,Z 370.613,A -85,B 0,C 180,E1 -21546.757,E2 -21546.757} C_VEL
LIN {X 0,Y 199.701,Z 370.606,A -85,B 0,C 180,E1 -21549.307,E2 -21549.307} C_VEL
LIN {X 0,Y 199.665,Z 370.612,A -85,B 0,C 180,E1 -21552.339,E2 -21552.339} C_VEL
LIN {X 0,Y 199.633,Z 370.617,A -85,B 0,C 180,E1 -21555.244,E2 -21555.244} C_VEL
LIN {X 0,Y 199.6,Z 370.618,A -85,B 0,C 180,E1 -21558.011,E2 -21558.011} C_VEL
LIN {X 0,Y 199.616,Z 370.619,A -85,B 0,C 180,E1 -21560.767,E2 -21560.767} C_VEL
LIN {X 0,Y 199.615,Z 370.615,A -85,B 0,C 180,E1 -21565.714,E2 -21565.714} C_VEL
LIN {X 0,Y 199.703,Z 370.607,A -85,B 0,C 180,E1 -21568.138,E2 -21568.138} C_VEL
LIN {X 0,Y 199.69,Z 370.61,A -85,B 0,C 180,E1 -21572.773,E2 -21572.773} C_VEL
LIN {X 0,Y 199.741,Z 370.604,A -85,B 0,C 180,E1 -21577.23,E2 -21577.23} C_VEL
LIN {X 0,Y 199.84,Z 370.588,A -85,B 0,C 180,E1 -21581.722,E2 -21581.722} C_VEL
LIN {X 0,Y 199.852,Z 370.588,A -85,B 0,C 180,E1 -21585.75,E2 -21585.75} C_VEL
LIN {X 0,Y 200.079,Z 370.559,A -85,B 0,C 180,E1 -21589.885,E2 -21589.885} C_VEL
LIN {X 0,Y 200.136,Z 370.55,A -85,B 0,C 180,E1 -21591.926,E2 -21591.926} C_VEL
LIN {X 0,Y 200.326,Z 370.53,A -85,B 0,C 180,E1 -21597.99,E2 -21597.99} C_VEL
LIN {X 0,Y 200.484,Z 370.508,A -85,B 0,C 180,E1 -21600,E2 -21600} C_VEL
LIN {X 0,Y 200.032,Z 370.568,A -85,B 0,C 180,E1 -21604.03,E2 -21604.03} C_VEL
LIN {X 0,Y 200.09,Z 370.559,A -85,B 0,C 180,E1 -21608.077,E2 -21608.077} C_VEL
LIN {X 0,Y 199.879,Z 370.588,A -85,B 0,C 180,E1 -21612.179,E2 -21612.179} C_VEL
LIN {X 0,Y 199.809,Z 370.593,A -85,B 0,C 180,E1 -21616.343,E2 -21616.343} C_VEL
LIN {X 0,Y 199.704,Z 370.608,A -85,B 0,C 180,E1 -21620.605,E2 -21620.605} C_VEL
LIN {X 0,Y 199.677,Z 370.607,A -85,B 0,C 180,E1 -21624.984,E2 -21624.984} C_VEL
LIN {X 0,Y 199.668,Z 370.613,A -85,B 0,C 180,E1 -21629.524,E2 -21629.524} C_VEL
LIN {X 0,Y 199.661,Z 370.612,A -85,B 0,C 180,E1 -21632.35,E2 -21632.35} C_VEL
LIN {X 0,Y 199.661,Z 370.612,A -85,B 0,C 180,E1 -21636.756,E2 -21636.756} C_VEL
LIN {X 0,Y 199.902,Z 370.692,A -85,B 0,C 180,E1 -21640.822,E2 -21640.822} C_VEL
LIN {X 0,Y 201.69,Z 379.567,A -85,B 0,C 180,E1 -21647.034,E2 -21647.034} C_VEL
LIN {X 0,Y 202.927,Z 384.931,A -85,B 0,C 180,E1 -21650.624,E2 -21650.624} C_VEL
LIN {X 0,Y 202.613,Z 388.428,A -85,B 0,C 180,E1 -21652.921,E2 -21652.921} C_VEL
LIN {X 0,Y 200.987,Z 395.649,A -85,B 0,C 180,E1 -21657.651,E2 -21657.651} C_VEL
LIN {X 0,Y 199.728,Z 403.382,A -85,B 0,C 180,E1 -21662.777,E2 -21662.777} C_VEL
LIN {X 0,Y 199.177,Z 408.352,A -85,B 0,C 180,E1 -21665.975,E2 -21665.975} C_VEL
LIN {X 0,Y 198.836,Z 421.946,A -85,B 0,C 180,E1 -21667.257,E2 -21667.257} C_VEL
LIN {X 0,Y 199.124,Z 434.388,A -85,B 0,C 180,E1 -21668.791,E2 -21668.791} C_VEL
LIN {X 0,Y 199.746,Z 446.906,A -85,B 0,C 180,E1 -21670.741,E2 -21670.741} C_VEL
LIN {X 0,Y 200.609,Z 458.49,A -85,B 0,C 180,E1 -21672.938,E2 -21672.938} C_VEL
LIN {X 0,Y 201.329,Z 466.82,A -85,B 0,C 180,E1 -21674.822,E2 -21674.822} C_VEL
LIN {X 0,Y 200.779,Z 475.88,A -85,B 0,C 180,E1 -21677.363,E2 -21677.363} C_VEL
LIN {X 0,Y 200.557,Z 484.745,A -85,B 0,C 180,E1 -21680.418,E2 -21680.418} C_VEL
LIN {X 0,Y 200.843,Z 491.919,A -85,B 0,C 180,E1 -21683.47,E2 -21683.47} C_VEL
LIN {X 0,Y 201.312,Z 496.677,A -85,B 0,C 180,E1 -21685.996,E2 -21685.996} C_VEL
LIN {X 0,Y 201.539,Z 498.493,A -85,B 0,C 180,E1 -21687.126,E2 -21687.126} C_VEL
LIN {X 0,Y 201.323,Z 499.892,A -85,B 0,C 180,E1 -21688.168,E2 -21688.168} C_VEL
LIN {X 0,Y 199.887,Z 501.364,A -85,B 0,C 180,E1 -21689.752,E2 -21689.752} C_VEL
LIN {X 0,Y 196.144,Z 502.745,A -85,B 0,C 180,E1 -21692.433,E2 -21692.433} C_VEL
LIN {X 0,Y 193.076,Z 503.683,A -85,B 0,C 180,E1 -21695.295,E2 -21695.295} C_VEL
LIN {X 0,Y 192.803,Z 503.866,A -85,B 0,C 180,E1 -21695.892,E2 -21695.892} C_VEL
LIN {X 0,Y 192.054,Z 504.638,A -85,B 0,C 180,E1 -21698.869,E2 -21698.869} C_VEL
LIN {X 0,Y 191.993,Z 504.723,A -85,B 0,C 180,E1 -21702.687,E2 -21702.687} C_VEL
LIN {X 0,Y 193.114,Z 503.692,A -85,B 0,C 180,E1 -21706.926,E2 -21706.926} C_VEL
LIN {X 0,Y 195.664,Z 501.519,A -85,B 0,C 180,E1 -21711.05,E2 -21711.05} C_VEL
LIN {X 0,Y 199.743,Z 498.234,A -85,B 0,C 180,E1 -21714.975,E2 -21714.975} C_VEL
LIN {X 0,Y 205.07,Z 493.791,A -85,B 0,C 180,E1 -21718.672,E2 -21718.672} C_VEL
LIN {X 0,Y 210.957,Z 488.185,A -85,B 0,C 180,E1 -21722.211,E2 -21722.211} C_VEL
LIN {X 0,Y 217.818,Z 481.459,A -85,B 0,C 180,E1 -21725.506,E2 -21725.506} C_VEL
LIN {X 0,Y 222.742,Z 475.754,A -85,B 0,C 180,E1 -21728.026,E2 -21728.026} C_VEL
LIN {X 0,Y 227.169,Z 470.024,A -85,B 0,C 180,E1 -21730.518,E2 -21730.518} C_VEL
LIN {X 0,Y 232.711,Z 462.356,A -85,B 0,C 180,E1 -21733.997,E2 -21733.997} C_VEL
LIN {X 0,Y 235.43,Z 458.665,A -85,B 0,C 180,E1 -21735.762,E2 -21735.762} C_VEL
LIN {X 0,Y 236.44,Z 457.002,A -85,B 0,C 180,E1 -21736.869,E2 -21736.869} C_VEL
LIN {X 0,Y 237.337,Z 454.372,A -85,B 0,C 180,E1 -21740.346,E2 -21740.346} C_VEL
LIN {X 0,Y 237.847,Z 453.409,A -85,B 0,C 180,E1 -21742.922,E2 -21742.922} C_VEL
LIN {X 0,Y 237.92,Z 453.277,A -85,B 0,C 180,E1 -21743.787,E2 -21743.787} C_VEL
LIN {X 0,Y 237.193,Z 453.874,A -85,B 0,C 180,E1 -21745.738,E2 -21745.738} C_VEL
LIN {X 0,Y 229.197,Z 459.035,A -85,B 0,C 180,E1 -21748.581,E2 -21748.581} C_VEL
LIN {X 0,Y 221.68,Z 462.914,A -85,B 0,C 180,E1 -21751.604,E2 -21751.604} C_VEL
LIN {X 0,Y 214.944,Z 465.357,A -85,B 0,C 180,E1 -21754.845,E2 -21754.845} C_VEL
LIN {X 0,Y 209.003,Z 466.471,A -85,B 0,C 180,E1 -21758.291,E2 -21758.291} C_VEL
LIN {X 0,Y 203.853,Z 466.292,A -85,B 0,C 180,E1 -21761.923,E2 -21761.923} C_VEL
LIN {X 0,Y 199.787,Z 464.678,A -85,B 0,C 180,E1 -21765.744,E2 -21765.744} C_VEL
LIN {X 0,Y 196.554,Z 461.712,A -85,B 0,C 180,E1 -21769.701,E2 -21769.701} C_VEL
LIN {X 0,Y 194.198,Z 457.309,A -85,B 0,C 180,E1 -21773.767,E2 -21773.767} C_VEL
LIN {X 0,Y 192.93,Z 451.322,A -85,B 0,C 180,E1 -21777.912,E2 -21777.912} C_VEL
LIN {X 0,Y 192.387,Z 444.68,A -85,B 0,C 180,E1 -21781.57,E2 -21781.57} C_VEL
LIN {X 0,Y 192.345,Z 436.428,A -85,B 0,C 180,E1 -21785.241,E2 -21785.241} C_VEL
LIN {X 0,Y 192.982,Z 427.917,A -85,B 0,C 180,E1 -21788.376,E2 -21788.376} C_VEL
LIN {X 0,Y 193.688,Z 418.554,A -85,B 0,C 180,E1 -21791.268,E2 -21791.268} C_VEL
LIN {X 0,Y 194.713,Z 407.424,A -85,B 0,C 180,E1 -21794.101,E2 -21794.101} C_VEL
LIN {X 0,Y 195.924,Z 395.154,A -85,B 0,C 180,E1 -21796.676,E2 -21796.676} C_VEL
LIN {X 0,Y 196.504,Z 389.452,A -85,B 0,C 180,E1 -21797.698,E2 -21797.698} C_VEL
LIN {X 0,Y 193.865,Z 376.689,A -85,B 0,C 180,E1 -21799.737,E2 -21799.737} C_VEL
LIN {X 0,Y 192.846,Z 371.462,A -85,B 0,C 180,E1 -21800.48,E2 -21800.48} C_VEL
LIN {X 0,Y 192.666,Z 371.482,A -85,B 0,C 180,E1 -21804.224,E2 -21804.224} C_VEL
LIN {X 0,Y 192.652,Z 371.488,A -85,B 0,C 180,E1 -21808.892,E2 -21808.892} C_VEL
LIN {X 0,Y 192.602,Z 371.49,A -85,B 0,C 180,E1 -21813.185,E2 -21813.185} C_VEL
LIN {X 0,Y 192.6,Z 371.493,A -85,B 0,C 180,E1 -21818.34,E2 -21818.34} C_VEL
LIN {X 0,Y 192.553,Z 371.497,A -85,B 0,C 180,E1 -21823.115,E2 -21823.115} C_VEL
LIN {X 0,Y 192.52,Z 371.505,A -85,B 0,C 180,E1 -21826.895,E2 -21826.895} C_VEL
LIN {X 0,Y 192.574,Z 371.491,A -85,B 0,C 180,E1 -21831.653,E2 -21831.653} C_VEL
LIN {X 0,Y 192.599,Z 371.493,A -85,B 0,C 180,E1 -21834.278,E2 -21834.278} C_VEL
LIN {X 0,Y 192.608,Z 371.488,A -85,B 0,C 180,E1 -21839.28,E2 -21839.28} C_VEL
LIN {X 0,Y 192.665,Z 371.482,A -85,B 0,C 180,E1 -21841.692,E2 -21841.692} C_VEL
LIN {X 0,Y 192.712,Z 371.48,A -85,B 0,C 180,E1 -21846.349,E2 -21846.349} C_VEL
LIN {X 0,Y 192.782,Z 371.469,A -85,B 0,C 180,E1 -21851.413,E2 -21851.413} C_VEL
LIN {X 0,Y 192.765,Z 371.47,A -85,B 0,C 180,E1 -21855.214,E2 -21855.214} C_VEL
LIN {X 0,Y 192.945,Z 371.449,A -85,B 0,C 180,E1 -21859.567,E2 -21859.567} C_VEL
LIN {X 0,Y 192.987,Z 371.445,A -85,B 0,C 180,E1 -21863.728,E2 -21863.728} C_VEL
LIN {X 0,Y 193.265,Z 371.41,A -85,B 0,C 180,E1 -21867.916,E2 -21867.916} C_VEL
LIN {X 0,Y 193.444,Z 371.39,A -85,B 0,C 180,E1 -21870,E2 -21870} C_VEL
LIN {X 0,Y 192.976,Z 371.443,A -85,B 0,C 180,E1 -21874.177,E2 -21874.177} C_VEL
LIN {X 0,Y 193.037,Z 371.439,A -85,B 0,C 180,E1 -21878.374,E2 -21878.374} C_VEL
LIN {X 0,Y 192.806,Z 371.462,A -85,B 0,C 180,E1 -21882.633,E2 -21882.633} C_VEL
LIN {X 0,Y 192.772,Z 371.471,A -85,B 0,C 180,E1 -21886.958,E2 -21886.958} C_VEL
LIN {X 0,Y 192.644,Z 371.485,A -85,B 0,C 180,E1 -21891.397,E2 -21891.397} C_VEL
LIN {X 0,Y 192.665,Z 371.484,A -85,B 0,C 180,E1 -21894.225,E2 -21894.225} C_VEL
LIN {X 0,Y 192.651,Z 371.484,A -85,B 0,C 180,E1 -21898.893,E2 -21898.893} C_VEL
LIN {X 0,Y 192.601,Z 371.493,A -85,B 0,C 180,E1 -21903.186,E2 -21903.186} C_VEL
LIN {X 0,Y 192.613,Z 371.486,A -85,B 0,C 180,E1 -21908.338,E2 -21908.338} C_VEL
LIN {X 0,Y 192.602,Z 371.495,A -85,B 0,C 180,E1 -21913.131,E2 -21913.131} C_VEL
LIN {X 0,Y 192.539,Z 371.498,A -85,B 0,C 180,E1 -21916.89,E2 -21916.89} C_VEL
LIN {X 0,Y 192.555,Z 371.499,A -85,B 0,C 180,E1 -21921.649,E2 -21921.649} C_VEL
LIN {X 0,Y 192.601,Z 371.49,A -85,B 0,C 180,E1 -21926.815,E2 -21926.815} C_VEL
LIN {X 0,Y 192.667,Z 371.483,A -85,B 0,C 180,E1 -21931.693,E2 -21931.693} C_VEL
LIN {X 0,Y 192.709,Z 371.478,A -85,B 0,C 180,E1 -21936.349,E2 -21936.349} C_VEL
LIN {X 0,Y 192.784,Z 371.467,A -85,B 0,C 180,E1 -21941.414,E2 -21941.414} C_VEL
LIN {X 0,Y 192.857,Z 371.461,A -85,B 0,C 180,E1 -21947.371,E2 -21947.371} C_VEL
LIN {X 0,Y 193.083,Z 371.428,A -85,B 0,C 180,E1 -21951.629,E2 -21951.629} C_VEL
LIN {X 0,Y 193.268,Z 371.409,A -85,B 0,C 180,E1 -21957.916,E2 -21957.916} C_VEL
LIN {X 0,Y 193.447,Z 371.384,A -85,B 0,C 180,E1 -21960,E2 -21960} C_VEL
LIN {X 0,Y 192.978,Z 371.447,A -85,B 0,C 180,E1 -21964.177,E2 -21964.177} C_VEL
LIN {X 0,Y 193.038,Z 371.436,A -85,B 0,C 180,E1 -21968.374,E2 -21968.374} C_VEL
LIN {X 0,Y 192.806,Z 371.468,A -85,B 0,C 180,E1 -21972.633,E2 -21972.633} C_VEL
LIN {X 0,Y 192.762,Z 371.468,A -85,B 0,C 180,E1 -21976.959,E2 -21976.959} C_VEL
LIN {X 0,Y 192.641,Z 371.488,A -85,B 0,C 180,E1 -21981.397,E2 -21981.397} C_VEL
LIN {X 0,Y 192.668,Z 371.483,A -85,B 0,C 180,E1 -21984.225,E2 -21984.225} C_VEL
LIN {X 0,Y 192.647,Z 371.486,A -85,B 0,C 180,E1 -21988.889,E2 -21988.889} C_VEL
LIN {X 0,Y 192.601,Z 371.49,A -85,B 0,C 180,E1 -21993.186,E2 -21993.186} C_VEL
LIN {X 0,Y 192.656,Z 371.486,A -85,B 0,C 180,E1 -21998.328,E2 -21998.328} C_VEL
LIN {X 0,Y 192.906,Z 371.609,A -85,B 0,C 180,E1 -22000.979,E2 -22000.979} C_VEL
LIN {X 0,Y 194.85,Z 381.022,A -85,B 0,C 180,E1 -22007.759,E2 -22007.759} C_VEL
LIN {X 0,Y 195.86,Z 385.794,A -85,B 0,C 180,E1 -22011.086,E2 -22011.086} C_VEL
LIN {X 0,Y 195.23,Z 389.446,A -85,B 0,C 180,E1 -22013.56,E2 -22013.56} C_VEL
LIN {X 0,Y 193.697,Z 396.296,A -85,B 0,C 180,E1 -22018.257,E2 -22018.257} C_VEL
LIN {X 0,Y 192.405,Z 404.538,A -85,B 0,C 180,E1 -22024.003,E2 -22024.003} C_VEL
LIN {X 0,Y 192.154,Z 407.334,A -85,B 0,C 180,E1 -22025.846,E2 -22025.846} C_VEL
LIN {X 0,Y 191.776,Z 420.005,A -85,B 0,C 180,E1 -22027.084,E2 -22027.084} C_VEL
LIN {X 0,Y 192.018,Z 433.511,A -85,B 0,C 180,E1 -22028.811,E2 -22028.811} C_VEL
LIN {X 0,Y 192.712,Z 446.953,A -85,B 0,C 180,E1 -22031.013,E2 -22031.013} C_VEL
LIN {X 0,Y 193.668,Z 458.755,A -85,B 0,C 180,E1 -22033.395,E2 -22033.395} C_VEL
LIN {X 0,Y 194.283,Z 466.814,A -85,B 0,C 180,E1 -22035.332,E2 -22035.332} C_VEL
LIN {X 0,Y 193.79,Z 476.596,A -85,B 0,C 180,E1 -22038.291,E2 -22038.291} C_VEL
LIN {X 0,Y 193.74,Z 484.289,A -85,B 0,C 180,E1 -22041.131,E2 -22041.131} C_VEL
LIN {X 0,Y 194.106,Z 491.25,A -85,B 0,C 180,E1 -22044.285,E2 -22044.285} C_VEL
LIN {X 0,Y 194.756,Z 496.716,A -85,B 0,C 180,E1 -22047.459,E2 -22047.459} C_VEL
LIN {X 0,Y 195.175,Z 500.108,A -85,B 0,C 180,E1 -22050,E2 -22050} C_VEL
LIN {X 0,Y 194.353,Z 501.878,A -85,B 0,C 180,E1 -22052.072,E2 -22052.072} C_VEL
LIN {X 0,Y 192.803,Z 503.866,A -85,B 0,C 180,E1 -22055.892,E2 -22055.892} C_VEL
LIN {X 0,Y 191.685,Z 504.285,A -85,B 0,C 180,E1 -22057.613,E2 -22057.613} C_VEL
LIN {X 0,Y 188.495,Z 504.021,A -85,B 0,C 180,E1 -22060.44,E2 -22060.44} C_VEL
LIN {X 0,Y 186.184,Z 503.437,A -85,B 0,C 180,E1 -22062.765,E2 -22062.765} C_VEL
LIN {X 0,Y 185.446,Z 503.062,A -85,B 0,C 180,E1 -22064.575,E2 -22064.575} C_VEL
LIN {X 0,Y 185.505,Z 502.96,A -85,B 0,C 180,E1 -22065.184,E2 -22065.184} C_VEL
LIN {X 0,Y 187.487,Z 501.644,A -85,B 0,C 180,E1 -22069.717,E2 -22069.717} C_VEL
LIN {X 0,Y 191.046,Z 499.273,A -85,B 0,C 180,E1 -22073.87,E2 -22073.87} C_VEL
LIN {X 0,Y 195.957,Z 495.795,A -85,B 0,C 180,E1 -22077.791,E2 -22077.791} C_VEL
LIN {X 0,Y 201.788,Z 491.194,A -85,B 0,C 180,E1 -22081.496,E2 -22081.496} C_VEL
LIN {X 0,Y 208.498,Z 485.502,A -85,B 0,C 180,E1 -22084.962,E2 -22084.962} C_VEL
LIN {X 0,Y 213.871,Z 480.537,A -85,B 0,C 180,E1 -22087.44,E2 -22087.44} C_VEL
LIN {X 0,Y 220.365,Z 473.462,A -85,B 0,C 180,E1 -22090.829,E2 -22090.829} C_VEL
LIN {X 0,Y 225.614,Z 467.133,A -85,B 0,C 180,E1 -22093.9,E2 -22093.9} C_VEL
LIN {X 0,Y 229.249,Z 462.813,A -85,B 0,C 180,E1 -22096.09,E2 -22096.09} C_VEL
LIN {X 0,Y 230.462,Z 461.234,A -85,B 0,C 180,E1 -22097.045,E2 -22097.045} C_VEL
LIN {X 0,Y 230.917,Z 460.285,A -85,B 0,C 180,E1 -22097.965,E2 -22097.965} C_VEL
LIN {X 0,Y 231.566,Z 458.567,A -85,B 0,C 180,E1 -22100.405,E2 -22100.405} C_VEL
LIN {X 0,Y 232.003,Z 457.565,A -85,B 0,C 180,E1 -22102.709,E2 -22102.709} C_VEL
LIN {X 0,Y 231.585,Z 457.55,A -85,B 0,C 180,E1 -22104.788,E2 -22104.788} C_VEL
LIN {X 0,Y 229.947,Z 458.519,A -85,B 0,C 180,E1 -22105.568,E2 -22105.568} C_VEL
LIN {X 0,Y 223.64,Z 461.987,A -85,B 0,C 180,E1 -22107.708,E2 -22107.708} C_VEL
LIN {X 0,Y 215.815,Z 465.372,A -85,B 0,C 180,E1 -22110.759,E2 -22110.759} C_VEL
LIN {X 0,Y 208.802,Z 467.415,A -85,B 0,C 180,E1 -22114.051,E2 -22114.051} C_VEL
LIN {X 0,Y 202.624,Z 468.11,A -85,B 0,C 180,E1 -22117.571,E2 -22117.571} C_VEL
LIN {X 0,Y 197.242,Z 467.52,A -85,B 0,C 180,E1 -22121.295,E2 -22121.295} C_VEL
LIN {X 0,Y 192.969,Z 465.576,A -85,B 0,C 180,E1 -22125.229,E2 -22125.229} C_VEL
LIN {X 0,Y 189.592,Z 462.236,A -85,B 0,C 180,E1 -22129.318,E2 -22129.318} C_VEL
LIN {X 0,Y 187.144,Z 457.469,A -85,B 0,C 180,E1 -22133.531,E2 -22133.531} C_VEL
LIN {X 0,Y 186.136,Z 452.866,A -85,B 0,C 180,E1 -22136.753,E2 -22136.753} C_VEL
LIN {X 0,Y 185.452,Z 446.293,A -85,B 0,C 180,E1 -22140.542,E2 -22140.542} C_VEL
LIN {X 0,Y 185.273,Z 438.165,A -85,B 0,C 180,E1 -22144.351,E2 -22144.351} C_VEL
LIN {X 0,Y 185.838,Z 428.246,A -85,B 0,C 180,E1 -22148.153,E2 -22148.153} C_VEL
LIN {X 0,Y 186.446,Z 419.733,A -85,B 0,C 180,E1 -22150.863,E2 -22150.863} C_VEL
LIN {X 0,Y 187.549,Z 408.618,A -85,B 0,C 180,E1 -22153.821,E2 -22153.821} C_VEL
LIN {X 0,Y 188.673,Z 396.409,A -85,B 0,C 180,E1 -22156.5,E2 -22156.5} C_VEL
LIN {X 0,Y 189.328,Z 389.188,A -85,B 0,C 180,E1 -22157.833,E2 -22157.833} C_VEL
LIN {X 0,Y 186.502,Z 375.971,A -85,B 0,C 180,E1 -22159.968,E2 -22159.968} C_VEL
LIN {X 0,Y 185.802,Z 372.339,A -85,B 0,C 180,E1 -22160.552,E2 -22160.552} C_VEL
LIN {X 0,Y 185.602,Z 372.363,A -85,B 0,C 180,E1 -22164.662,E2 -22164.662} C_VEL
LIN {X 0,Y 185.58,Z 372.368,A -85,B 0,C 180,E1 -22169.492,E2 -22169.492} C_VEL
LIN {X 0,Y 185.522,Z 372.371,A -85,B 0,C 180,E1 -22174.627,E2 -22174.627} C_VEL
LIN {X 0,Y 185.569,Z 372.369,A -85,B 0,C 180,E1 -22177.313,E2 -22177.313} C_VEL
LIN {X 0,Y 185.523,Z 372.375,A -85,B 0,C 180,E1 -22180.743,E2 -22180.743} C_VEL
LIN {X 0,Y 185.49,Z 372.378,A -85,B 0,C 180,E1 -22186.045,E2 -22186.045} C_VEL
LIN {X 0,Y 185.49,Z 372.376,A -85,B 0,C 180,E1 -22189.901,E2 -22189.901} C_VEL
LIN {X 0,Y 185.544,Z 372.371,A -85,B 0,C 180,E1 -22192.696,E2 -22192.696} C_VEL
LIN {X 0,Y 185.546,Z 372.371,A -85,B 0,C 180,E1 -22197.975,E2 -22197.975} C_VEL
LIN {X 0,Y 185.582,Z 372.365,A -85,B 0,C 180,E1 -22200.576,E2 -22200.576} C_VEL
LIN {X 0,Y 185.606,Z 372.363,A -85,B 0,C 180,E1 -22205.385,E2 -22205.385} C_VEL
LIN {X 0,Y 185.711,Z 372.35,A -85,B 0,C 180,E1 -22211.101,E2 -22211.101} C_VEL
LIN {X 0,Y 185.7,Z 372.352,A -85,B 0,C 180,E1 -22214.638,E2 -22214.638} C_VEL
LIN {X 0,Y 185.889,Z 372.327,A -85,B 0,C 180,E1 -22219.418,E2 -22219.418} C_VEL
LIN {X 0,Y 185.949,Z 372.321,A -85,B 0,C 180,E1 -22223.49,E2 -22223.49} C_VEL
LIN {X 0,Y 186.208,Z 372.288,A -85,B 0,C 180,E1 -22227.837,E2 -22227.837} C_VEL
LIN {X 0,Y 186.408,Z 372.267,A -85,B 0,C 180,E1 -22230,E2 -22230} C_VEL
LIN {X 0,Y 185.923,Z 372.322,A -85,B 0,C 180,E1 -22234.336,E2 -22234.336} C_VEL
LIN {X 0,Y 185.984,Z 372.317,A -85,B 0,C 180,E1 -22238.694,E2 -22238.694} C_VEL
LIN {X 0,Y 185.732,Z 372.343,A -85,B 0,C 180,E1 -22243.123,E2 -22243.123} C_VEL
LIN {X 0,Y 185.718,Z 372.353,A -85,B 0,C 180,E1 -22247.622,E2 -22247.622} C_VEL
LIN {X 0,Y 185.601,Z 372.362,A -85,B 0,C 180,E1 -22252.251,E2 -22252.251} C_VEL
LIN {X 0,Y 185.564,Z 372.37,A -85,B 0,C 180,E1 -22257.032,E2 -22257.032} C_VEL
LIN {X 0,Y 185.58,Z 372.365,A -85,B 0,C 180,E1 -22259.493,E2 -22259.493} C_VEL
LIN {X 0,Y 185.522,Z 372.374,A -85,B 0,C 180,E1 -22264.628,E2 -22264.628} C_VEL
LIN {X 0,Y 185.569,Z 372.367,A -85,B 0,C 180,E1 -22267.314,E2 -22267.314} C_VEL
LIN {X 0,Y 185.573,Z 372.367,A -85,B 0,C 180,E1 -22270.761,E2 -22270.761} C_VEL
LIN {X 0,Y 185.556,Z 372.37,A -85,B 0,C 180,E1 -22273.976,E2 -22273.976} C_VEL
LIN {X 0,Y 185.482,Z 372.38,A -85,B 0,C 180,E1 -22279.272,E2 -22279.272} C_VEL
LIN {X 0,Y 185.509,Z 372.377,A -85,B 0,C 180,E1 -22282.711,E2 -22282.711} C_VEL
LIN {X 0,Y 185.548,Z 372.37,A -85,B 0,C 180,E1 -22287.976,E2 -22287.976} C_VEL
LIN {X 0,Y 185.584,Z 372.368,A -85,B 0,C 180,E1 -22290.576,E2 -22290.576} C_VEL
LIN {X 0,Y 185.59,Z 372.365,A -85,B 0,C 180,E1 -22295.383,E2 -22295.383} C_VEL
LIN {X 0,Y 185.697,Z 372.351,A -85,B 0,C 180,E1 -22301.116,E2 -22301.116} C_VEL
LIN {X 0,Y 185.732,Z 372.348,A -85,B 0,C 180,E1 -22304.641,E2 -22304.641} C_VEL
LIN {X 0,Y 185.946,Z 372.32,A -85,B 0,C 180,E1 -22309.329,E2 -22309.329} C_VEL
LIN {X 0,Y 185.973,Z 372.317,A -85,B 0,C 180,E1 -22313.491,E2 -22313.491} C_VEL
LIN {X 0,Y 186.212,Z 372.288,A -85,B 0,C 180,E1 -22317.837,E2 -22317.837} C_VEL
LIN {X 0,Y 186.411,Z 372.26,A -85,B 0,C 180,E1 -22320,E2 -22320} C_VEL
LIN {X 0,Y 185.924,Z 372.327,A -85,B 0,C 180,E1 -22324.336,E2 -22324.336} C_VEL
LIN {X 0,Y 185.985,Z 372.314,A -85,B 0,C 180,E1 -22328.694,E2 -22328.694} C_VEL
LIN {X 0,Y 185.733,Z 372.348,A -85,B 0,C 180,E1 -22333.123,E2 -22333.123} C_VEL
LIN {X 0,Y 185.694,Z 372.348,A -85,B 0,C 180,E1 -22337.625,E2 -22337.625} C_VEL
LIN {X 0,Y 185.601,Z 372.366,A -85,B 0,C 180,E1 -22342.251,E2 -22342.251} C_VEL
LIN {X 0,Y 185.564,Z 372.366,A -85,B 0,C 180,E1 -22347.032,E2 -22347.032} C_VEL
LIN {X 0,Y 185.581,Z 372.367,A -85,B 0,C 180,E1 -22349.493,E2 -22349.493} C_VEL
LIN {X 0,Y 185.524,Z 372.37,A -85,B 0,C 180,E1 -22354.627,E2 -22354.627} C_VEL
LIN {X 0,Y 185.749,Z 372.347,A -85,B 0,C 180,E1 -22360.032,E2 -22360.032} C_VEL
LIN {X 0,Y 185.845,Z 372.415,A -85,B 0,C 180,E1 -22361.073,E2 -22361.073} C_VEL
LIN {X 0,Y 187.673,Z 381.144,A -85,B 0,C 180,E1 -22367.618,E2 -22367.618} C_VEL
LIN {X 0,Y 188.699,Z 385.407,A -85,B 0,C 180,E1 -22370.716,E2 -22370.716} C_VEL
LIN {X 0,Y 188.535,Z 387.797,A -85,B 0,C 180,E1 -22372.409,E2 -22372.409} C_VEL
LIN {X 0,Y 186.99,Z 394.187,A -85,B 0,C 180,E1 -22376.976,E2 -22376.976} C_VEL
LIN {X 0,Y 185.559,Z 402.439,A -85,B 0,C 180,E1 -22382.967,E2 -22382.967} C_VEL
LIN {X 0,Y 185.156,Z 406.159,A -85,B 0,C 180,E1 -22385.715,E2 -22385.715} C_VEL
LIN {X 0,Y 184.686,Z 418.622,A -85,B 0,C 180,E1 -22386.991,E2 -22386.991} C_VEL
LIN {X 0,Y 184.902,Z 432.436,A -85,B 0,C 180,E1 -22388.833,E2 -22388.833} C_VEL
LIN {X 0,Y 185.641,Z 446.083,A -85,B 0,C 180,E1 -22391.166,E2 -22391.166} C_VEL
LIN {X 0,Y 186.622,Z 457.622,A -85,B 0,C 180,E1 -22393.594,E2 -22393.594} C_VEL
LIN {X 0,Y 187.343,Z 464.681,A -85,B 0,C 180,E1 -22395.332,E2 -22395.332} C_VEL
LIN {X 0,Y 186.941,Z 473.942,A -85,B 0,C 180,E1 -22398.158,E2 -22398.158} C_VEL
LIN {X 0,Y 186.906,Z 482.419,A -85,B 0,C 180,E1 -22401.349,E2 -22401.349} C_VEL
LIN {X 0,Y 187.343,Z 489.474,A -85,B 0,C 180,E1 -22404.618,E2 -22404.618} C_VEL
LIN {X 0,Y 188.026,Z 494.985,A -85,B 0,C 180,E1 -22407.858,E2 -22407.858} C_VEL
LIN {X 0,Y 188.388,Z 497.803,A -85,B 0,C 180,E1 -22410,E2 -22410} C_VEL
LIN {X 0,Y 187.569,Z 499.708,A -85,B 0,C 180,E1 -22412.147,E2 -22412.147} C_VEL
LIN {X 0,Y 185.795,Z 502.093,A -85,B 0,C 180,E1 -22416.516,E2 -22416.516} C_VEL
LIN {X 0,Y 184.998,Z 503.105,A -85,B 0,C 180,E1 -22420.95,E2 -22420.95} C_VEL
LIN {X 0,Y 185.505,Z 502.96,A -85,B 0,C 180,E1 -22425.184,E2 -22425.184} C_VEL
LIN {X 0,Y 185.433,Z 502.581,A -85,B 0,C 180,E1 -22427.007,E2 -22427.007} C_VEL
LIN {X 0,Y 184.125,Z 501.308,A -85,B 0,C 180,E1 -22430.031,E2 -22430.031} C_VEL
LIN {X 0,Y 183.564,Z 499.531,A -85,B 0,C 180,E1 -22433.053,E2 -22433.053} C_VEL
LIN {X 0,Y 184.642,Z 498.365,A -85,B 0,C 180,E1 -22434.815,E2 -22434.815} C_VEL
LIN {X 0,Y 189.714,Z 495.305,A -85,B 0,C 180,E1 -22438.789,E2 -22438.789} C_VEL
LIN {X 0,Y 195.746,Z 491.122,A -85,B 0,C 180,E1 -22442.585,E2 -22442.585} C_VEL
LIN {X 0,Y 202.736,Z 485.91,A -85,B 0,C 180,E1 -22446.109,E2 -22446.109} C_VEL
LIN {X 0,Y 208.28,Z 481.345,A -85,B 0,C 180,E1 -22448.627,E2 -22448.627} C_VEL
LIN {X 0,Y 213.405,Z 476.489,A -85,B 0,C 180,E1 -22451.198,E2 -22451.198} C_VEL
LIN {X 0,Y 218.25,Z 471.483,A -85,B 0,C 180,E1 -22453.815,E2 -22453.815} C_VEL
LIN {X 0,Y 222.901,Z 466.557,A -85,B 0,C 180,E1 -22456.484,E2 -22456.484} C_VEL
LIN {X 0,Y 224.331,Z 465.008,A -85,B 0,C 180,E1 -22457.411,E2 -22457.411} C_VEL
LIN {X 0,Y 225.084,Z 463.801,A -85,B 0,C 180,E1 -22458.537,E2 -22458.537} C_VEL
LIN {X 0,Y 225.792,Z 461.93,A -85,B 0,C 180,E1 -22461.499,E2 -22461.499} C_VEL
LIN {X 0,Y 225.646,Z 461.283,A -85,B 0,C 180,E1 -22464.077,E2 -22464.077} C_VEL
LIN {X 0,Y 222.437,Z 462.867,A -85,B 0,C 180,E1 -22465.339,E2 -22465.339} C_VEL
LIN {X 0,Y 213.955,Z 466.481,A -85,B 0,C 180,E1 -22468.293,E2 -22468.293} C_VEL
LIN {X 0,Y 206.233,Z 468.709,A -85,B 0,C 180,E1 -22471.504,E2 -22471.504} C_VEL
LIN {X 0,Y 199.364,Z 469.659,A -85,B 0,C 180,E1 -22474.974,E2 -22474.974} C_VEL
LIN {X 0,Y 193.321,Z 469.348,A -85,B 0,C 180,E1 -22478.682,E2 -22478.682} C_VEL
LIN {X 0,Y 188.273,Z 467.669,A -85,B 0,C 180,E1 -22482.624,E2 -22482.624} C_VEL
LIN {X 0,Y 184.309,Z 464.656,A -85,B 0,C 180,E1 -22486.774,E2 -22486.774} C_VEL
LIN {X 0,Y 181.257,Z 460.276,A -85,B 0,C 180,E1 -22491.077,E2 -22491.077} C_VEL
LIN {X 0,Y 179.287,Z 454.351,A -85,B 0,C 180,E1 -22495.503,E2 -22495.503} C_VEL
LIN {X 0,Y 178.521,Z 447.832,A -85,B 0,C 180,E1 -22499.436,E2 -22499.436} C_VEL
LIN {X 0,Y 178.153,Z 439.803,A -85,B 0,C 180,E1 -22503.392,E2 -22503.392} C_VEL
LIN {X 0,Y 178.563,Z 430.004,A -85,B 0,C 180,E1 -22507.349,E2 -22507.349} C_VEL
LIN {X 0,Y 179.227,Z 421.655,A -85,B 0,C 180,E1 -22510.163,E2 -22510.163} C_VEL
LIN {X 0,Y 180.337,Z 409.678,A -85,B 0,C 180,E1 -22513.522,E2 -22513.522} C_VEL
LIN {X 0,Y 181.479,Z 397.514,A -85,B 0,C 180,E1 -22516.306,E2 -22516.306} C_VEL
LIN {X 0,Y 182.194,Z 390.383,A -85,B 0,C 180,E1 -22517.684,E2 -22517.684} C_VEL
LIN {X 0,Y 179.808,Z 378.668,A -85,B 0,C 180,E1 -22519.676,E2 -22519.676} C_VEL
LIN {X 0,Y 178.769,Z 373.215,A -85,B 0,C 180,E1 -22520.515,E2 -22520.515} C_VEL
LIN {X 0,Y 178.514,Z 373.243,A -85,B 0,C 180,E1 -22525.662,E2 -22525.662} C_VEL
LIN {X 0,Y 178.502,Z 373.251,A -85,B 0,C 180,E1 -22530.786,E2 -22530.786} C_VEL
LIN {X 0,Y 178.486,Z 373.246,A -85,B 0,C 180,E1 -22534.219,E2 -22534.219} C_VEL
LIN {X 0,Y 178.467,Z 373.255,A -85,B 0,C 180,E1 -22539.055,E2 -22539.055} C_VEL
LIN {X 0,Y 178.439,Z 373.254,A -85,B 0,C 180,E1 -22542.033,E2 -22542.033} C_VEL
LIN {X 0,Y 178.426,Z 373.259,A -85,B 0,C 180,E1 -22545.153,E2 -22545.153} C_VEL
LIN {X 0,Y 178.417,Z 373.261,A -85,B 0,C 180,E1 -22548.454,E2 -22548.454} C_VEL
LIN {X 0,Y 178.45,Z 373.254,A -85,B 0,C 180,E1 -22553.789,E2 -22553.789} C_VEL
LIN {X 0,Y 178.491,Z 373.252,A -85,B 0,C 180,E1 -22556.548,E2 -22556.548} C_VEL
LIN {X 0,Y 178.523,Z 373.243,A -85,B 0,C 180,E1 -22560.006,E2 -22560.006} C_VEL
LIN {X 0,Y 178.535,Z 373.245,A -85,B 0,C 180,E1 -22564.875,E2 -22564.875} C_VEL
LIN {X 0,Y 178.655,Z 373.23,A -85,B 0,C 180,E1 -22570.755,E2 -22570.755} C_VEL
LIN {X 0,Y 178.66,Z 373.226,A -85,B 0,C 180,E1 -22576.348,E2 -22576.348} C_VEL
LIN {X 0,Y 178.912,Z 373.198,A -85,B 0,C 180,E1 -22580.96,E2 -22580.96} C_VEL
LIN {X 0,Y 179.154,Z 373.167,A -85,B 0,C 180,E1 -22587.752,E2 -22587.752} C_VEL
LIN {X 0,Y 179.371,Z 373.143,A -85,B 0,C 180,E1 -22590,E2 -22590} C_VEL
LIN {X 0,Y 178.87,Z 373.199,A -85,B 0,C 180,E1 -22594.507,E2 -22594.507} C_VEL
LIN {X 0,Y 178.912,Z 373.198,A -85,B 0,C 180,E1 -22599.04,E2 -22599.04} C_VEL
LIN {X 0,Y 178.661,Z 373.226,A -85,B 0,C 180,E1 -22603.652,E2 -22603.652} C_VEL
LIN {X 0,Y 178.639,Z 373.232,A -85,B 0,C 180,E1 -22609.231,E2 -22609.231} C_VEL
LIN {X 0,Y 178.535,Z 373.245,A -85,B 0,C 180,E1 -22615.125,E2 -22615.125} C_VEL
LIN {X 0,Y 178.48,Z 373.247,A -85,B 0,C 180,E1 -22620.791,E2 -22620.791} C_VEL
LIN {X 0,Y 178.486,Z 373.251,A -85,B 0,C 180,E1 -22624.22,E2 -22624.22} C_VEL
LIN {X 0,Y 178.482,Z 373.248,A -85,B 0,C 180,E1 -22629.053,E2 -22629.053} C_VEL
LIN {X 0,Y 178.502,Z 373.249,A -85,B 0,C 180,E1 -22632.016,E2 -22632.016} C_VEL
LIN {X 0,Y 178.458,Z 373.255,A -85,B 0,C 180,E1 -22635.144,E2 -22635.144} C_VEL
LIN {X 0,Y 178.419,Z 373.256,A -85,B 0,C 180,E1 -22638.454,E2 -22638.454} C_VEL
LIN {X 0,Y 178.425,Z 373.256,A -85,B 0,C 180,E1 -22643.784,E2 -22643.784} C_VEL
LIN {X 0,Y 178.489,Z 373.247,A -85,B 0,C 180,E1 -22646.548,E2 -22646.548} C_VEL
LIN {X 0,Y 178.525,Z 373.246,A -85,B 0,C 180,E1 -22650.007,E2 -22650.007} C_VEL
LIN {X 0,Y 178.537,Z 373.242,A -85,B 0,C 180,E1 -22654.876,E2 -22654.876} C_VEL
LIN {X 0,Y 178.641,Z 373.232,A -85,B 0,C 180,E1 -22660.77,E2 -22660.77} C_VEL
LIN {X 0,Y 178.679,Z 373.224,A -85,B 0,C 180,E1 -22664.019,E2 -22664.019} C_VEL
LIN {X 0,Y 178.898,Z 373.198,A -85,B 0,C 180,E1 -22669.154,E2 -22669.154} C_VEL
LIN {X 0,Y 178.938,Z 373.194,A -85,B 0,C 180,E1 -22673.234,E2 -22673.234} C_VEL
LIN {X 0,Y 179.158,Z 373.166,A -85,B 0,C 180,E1 -22677.752,E2 -22677.752} C_VEL
LIN {X 0,Y 179.374,Z 373.137,A -85,B 0,C 180,E1 -22680,E2 -22680} C_VEL
LIN {X 0,Y 178.871,Z 373.205,A -85,B 0,C 180,E1 -22684.507,E2 -22684.507} C_VEL
LIN {X 0,Y 178.914,Z 373.194,A -85,B 0,C 180,E1 -22689.041,E2 -22689.041} C_VEL
LIN {X 0,Y 178.662,Z 373.229,A -85,B 0,C 180,E1 -22693.652,E2 -22693.652} C_VEL
LIN {X 0,Y 178.627,Z 373.232,A -85,B 0,C 180,E1 -22699.217,E2 -22699.217} C_VEL
LIN {X 0,Y 178.538,Z 373.24,A -85,B 0,C 180,E1 -22705.124,E2 -22705.124} C_VEL
LIN {X 0,Y 178.48,Z 373.251,A -85,B 0,C 180,E1 -22710.791,E2 -22710.791} C_VEL
LIN {X 0,Y 178.487,Z 373.248,A -85,B 0,C 180,E1 -22714.219,E2 -22714.219} C_VEL
LIN {X 0,Y 178.728,Z 373.22,A -85,B 0,C 180,E1 -22720.376,E2 -22720.376} C_VEL
LIN {X 0,Y 178.855,Z 373.305,A -85,B 0,C 180,E1 -22721.302,E2 -22721.302} C_VEL
LIN {X 0,Y 180.576,Z 381.497,A -85,B 0,C 180,E1 -22727.687,E2 -22727.687} C_VEL
LIN {X 0,Y 181.574,Z 385.525,A -85,B 0,C 180,E1 -22730.726,E2 -22730.726} C_VEL
LIN {X 0,Y 181.158,Z 388.629,A -85,B 0,C 180,E1 -22733.035,E2 -22733.035} C_VEL
LIN {X 0,Y 179.555,Z 395.371,A -85,B 0,C 180,E1 -22738.102,E2 -22738.102} C_VEL
LIN {X 0,Y 178.26,Z 403.446,A -85,B 0,C 180,E1 -22744.298,E2 -22744.298} C_VEL
LIN {X 0,Y 178.134,Z 405.184,A -85,B 0,C 180,E1 -22745.624,E2 -22745.624} C_VEL
LIN {X 0,Y 177.604,Z 417.882,A -85,B 0,C 180,E1 -22746.997,E2 -22746.997} C_VEL
LIN {X 0,Y 177.813,Z 431.198,A -85,B 0,C 180,E1 -22748.859,E2 -22748.859} C_VEL
LIN {X 0,Y 178.552,Z 444.057,A -85,B 0,C 180,E1 -22751.133,E2 -22751.133} C_VEL
LIN {X 0,Y 179.595,Z 456.376,A -85,B 0,C 180,E1 -22753.81,E2 -22753.81} C_VEL
LIN {X 0,Y 180.392,Z 464.469,A -85,B 0,C 180,E1 -22755.907,E2 -22755.907} C_VEL
LIN {X 0,Y 180.071,Z 474.789,A -85,B 0,C 180,E1 -22759.316,E2 -22759.316} C_VEL
LIN {X 0,Y 180.21,Z 483.055,A -85,B 0,C 180,E1 -22762.718,E2 -22762.718} C_VEL
LIN {X 0,Y 180.666,Z 488.653,A -85,B 0,C 180,E1 -22765.538,E2 -22765.538} C_VEL
LIN {X 0,Y 181.406,Z 493.983,A -85,B 0,C 180,E1 -22768.89,E2 -22768.89} C_VEL
LIN {X 0,Y 181.597,Z 495.404,A -85,B 0,C 180,E1 -22770,E2 -22770} C_VEL
LIN {X 0,Y 180.796,Z 497.467,A -85,B 0,C 180,E1 -22772.228,E2 -22772.228} C_VEL
LIN {X 0,Y 178.927,Z 500.071,A -85,B 0,C 180,E1 -22776.767,E2 -22776.767} C_VEL
LIN {X 0,Y 178.135,Z 501.313,A -85,B 0,C 180,E1 -22781.377,E2 -22781.377} C_VEL
LIN {X 0,Y 178.754,Z 501.411,A -85,B 0,C 180,E1 -22785.975,E2 -22785.975} C_VEL
LIN {X 0,Y 180.842,Z 500.427,A -85,B 0,C 180,E1 -22790.473,E2 -22790.473} C_VEL
LIN {X 0,Y 184.642,Z 498.365,A -85,B 0,C 180,E1 -22794.815,E2 -22794.815} C_VEL
LIN {X 0,Y 185.957,Z 497.184,A -85,B 0,C 180,E1 -22796.557,E2 -22796.557} C_VEL
LIN {X 0,Y 186.818,Z 494.875,A -85,B 0,C 180,E1 -22799.517,E2 -22799.517} C_VEL
LIN {X 0,Y 187.76,Z 492.852,A -85,B 0,C 180,E1 -22801.85,E2 -22801.85} C_VEL
LIN {X 0,Y 189.428,Z 491.205,A -85,B 0,C 180,E1 -22803.498,E2 -22803.498} C_VEL
LIN {X 0,Y 190.263,Z 490.624,A -85,B 0,C 180,E1 -22804.008,E2 -22804.008} C_VEL
LIN {X 0,Y 199.029,Z 484.843,A -85,B 0,C 180,E1 -22808.167,E2 -22808.167} C_VEL
LIN {X 0,Y 205.56,Z 479.73,A -85,B 0,C 180,E1 -22811.221,E2 -22811.221} C_VEL
LIN {X 0,Y 211.518,Z 474.442,A -85,B 0,C 180,E1 -22814.248,E2 -22814.248} C_VEL
LIN {X 0,Y 216.668,Z 469.63,A -85,B 0,C 180,E1 -22817.064,E2 -22817.064} C_VEL
LIN {X 0,Y 218.004,Z 468.382,A -85,B 0,C 180,E1 -22817.857,E2 -22817.857} C_VEL
LIN {X 0,Y 218.979,Z 467.209,A -85,B 0,C 180,E1 -22818.881,E2 -22818.881} C_VEL
LIN {X 0,Y 219.304,Z 466.26,A -85,B 0,C 180,E1 -22820.276,E2 -22820.276} C_VEL
LIN {X 0,Y 219.53,Z 464.955,A -85,B 0,C 180,E1 -22823.164,E2 -22823.164} C_VEL
LIN {X 0,Y 217.074,Z 465.877,A -85,B 0,C 180,E1 -22824.354,E2 -22824.354} C_VEL
LIN {X 0,Y 208.307,Z 468.981,A -85,B 0,C 180,E1 -22827.328,E2 -22827.328} C_VEL
LIN {X 0,Y 200.295,Z 470.792,A -85,B 0,C 180,E1 -22830.578,E2 -22830.578} C_VEL
LIN {X 0,Y 193.135,Z 471.299,A -85,B 0,C 180,E1 -22834.108,E2 -22834.108} C_VEL
LIN {X 0,Y 186.833,Z 470.565,A -85,B 0,C 180,E1 -22837.903,E2 -22837.903} C_VEL
LIN {X 0,Y 181.56,Z 468.531,A -85,B 0,C 180,E1 -22841.96,E2 -22841.96} C_VEL
LIN {X 0,Y 177.42,Z 465.122,A -85,B 0,C 180,E1 -22846.25,E2 -22846.25} C_VEL
LIN {X 0,Y 174.247,Z 460.35,A -85,B 0,C 180,E1 -22850.715,E2 -22850.715} C_VEL
LIN {X 0,Y 172.226,Z 454.075,A -85,B 0,C 180,E1 -22855.318,E2 -22855.318} C_VEL
LIN {X 0,Y 171.373,Z 446.092,A -85,B 0,C 180,E1 -22860,E2 -22860} C_VEL
LIN {X 0,Y 171.128,Z 437.426,A -85,B 0,C 180,E1 -22864.121,E2 -22864.121} C_VEL
LIN {X 0,Y 171.726,Z 426.902,A -85,B 0,C 180,E1 -22868.235,E2 -22868.235} C_VEL
LIN {X 0,Y 172.583,Z 415.85,A -85,B 0,C 180,E1 -22871.748,E2 -22871.748} C_VEL
LIN {X 0,Y 173.624,Z 404.823,A -85,B 0,C 180,E1 -22874.654,E2 -22874.654} C_VEL
LIN {X 0,Y 174.839,Z 392.872,A -85,B 0,C 180,E1 -22877.244,E2 -22877.244} C_VEL
LIN {X 0,Y 175.002,Z 389.831,A -85,B 0,C 180,E1 -22877.831,E2 -22877.831} C_VEL
LIN {X 0,Y 172.141,Z 376.334,A -85,B 0,C 180,E1 -22880.111,E2 -22880.111} C_VEL
LIN {X 0,Y 171.752,Z 374.089,A -85,B 0,C 180,E1 -22880.465,E2 -22880.465} C_VEL
LIN {X 0,Y 171.42,Z 374.128,A -85,B 0,C 180,E1 -22886.807,E2 -22886.807} C_VEL
LIN {X 0,Y 171.459,Z 374.127,A -85,B 0,C 180,E1 -22890.596,E2 -22890.596} C_VEL
LIN {X 0,Y 171.405,Z 374.13,A -85,B 0,C 180,E1 -22895.031,E2 -22895.031} C_VEL
LIN {X 0,Y 171.422,Z 374.133,A -85,B 0,C 180,E1 -22898.834,E2 -22898.834} C_VEL
LIN {X 0,Y 171.352,Z 374.136,A -85,B 0,C 180,E1 -22904.207,E2 -22904.207} C_VEL
LIN {X 0,Y 171.349,Z 374.139,A -85,B 0,C 180,E1 -22908.985,E2 -22908.985} C_VEL
LIN {X 0,Y 171.414,Z 374.127,A -85,B 0,C 180,E1 -22912.048,E2 -22912.048} C_VEL
LIN {X 0,Y 171.411,Z 374.133,A -85,B 0,C 180,E1 -22915.086,E2 -22915.086} C_VEL
LIN {X 0,Y 171.45,Z 374.125,A -85,B 0,C 180,E1 -22920.534,E2 -22920.534} C_VEL
LIN {X 0,Y 171.466,Z 374.125,A -85,B 0,C 180,E1 -22925.803,E2 -22925.803} C_VEL
LIN {X 0,Y 171.611,Z 374.107,A -85,B 0,C 180,E1 -22930.875,E2 -22930.875} C_VEL
LIN {X 0,Y 171.581,Z 374.11,A -85,B 0,C 180,E1 -22935.773,E2 -22935.773} C_VEL
LIN {X 0,Y 171.848,Z 374.079,A -85,B 0,C 180,E1 -22940.585,E2 -22940.585} C_VEL
LIN {X 0,Y 171.818,Z 374.077,A -85,B 0,C 180,E1 -22945.308,E2 -22945.308} C_VEL
LIN {X 0,Y 172.334,Z 374.02,A -85,B 0,C 180,E1 -22950,E2 -22950} C_VEL
LIN {X 0,Y 171.818,Z 374.077,A -85,B 0,C 180,E1 -22954.693,E2 -22954.693} C_VEL
LIN {X 0,Y 171.849,Z 374.079,A -85,B 0,C 180,E1 -22959.415,E2 -22959.415} C_VEL
LIN {X 0,Y 171.581,Z 374.11,A -85,B 0,C 180,E1 -22964.227,E2 -22964.227} C_VEL
LIN {X 0,Y 171.559,Z 374.114,A -85,B 0,C 180,E1 -22969.575,E2 -22969.575} C_VEL
LIN {X 0,Y 171.47,Z 374.127,A -85,B 0,C 180,E1 -22975.617,E2 -22975.617} C_VEL
LIN {X 0,Y 171.443,Z 374.124,A -85,B 0,C 180,E1 -22980.587,E2 -22980.587} C_VEL
LIN {X 0,Y 171.409,Z 374.133,A -85,B 0,C 180,E1 -22985.031,E2 -22985.031} C_VEL
LIN {X 0,Y 171.435,Z 374.125,A -85,B 0,C 180,E1 -22988.84,E2 -22988.84} C_VEL
LIN {X 0,Y 171.388,Z 374.134,A -85,B 0,C 180,E1 -22994.196,E2 -22994.196} C_VEL
LIN {X 0,Y 171.348,Z 374.139,A -85,B 0,C 180,E1 -22998.986,E2 -22998.986} C_VEL
LIN {X 0,Y 171.391,Z 374.134,A -85,B 0,C 180,E1 -23002.042,E2 -23002.042} C_VEL
LIN {X 0,Y 171.4,Z 374.131,A -85,B 0,C 180,E1 -23005.093,E2 -23005.093} C_VEL
LIN {X 0,Y 171.452,Z 374.128,A -85,B 0,C 180,E1 -23010.535,E2 -23010.535} C_VEL
LIN {X 0,Y 171.461,Z 374.124,A -85,B 0,C 180,E1 -23015.803,E2 -23015.803} C_VEL
LIN {X 0,Y 171.598,Z 374.108,A -85,B 0,C 180,E1 -23020.874,E2 -23020.874} C_VEL
LIN {X 0,Y 171.616,Z 374.106,A -85,B 0,C 180,E1 -23025.777,E2 -23025.777} C_VEL
LIN {X 0,Y 171.914,Z 374.067,A -85,B 0,C 180,E1 -23030.589,E2 -23030.589} C_VEL
LIN {X 0,Y 171.829,Z 374.08,A -85,B 0,C 180,E1 -23035.308,E2 -23035.308} C_VEL
LIN {X 0,Y 172.337,Z 374.013,A -85,B 0,C 180,E1 -23040,E2 -23040} C_VEL
LIN {X 0,Y 171.819,Z 374.082,A -85,B 0,C 180,E1 -23044.693,E2 -23044.693} C_VEL
LIN {X 0,Y 171.85,Z 374.073,A -85,B 0,C 180,E1 -23049.415,E2 -23049.415} C_VEL
LIN {X 0,Y 171.58,Z 374.113,A -85,B 0,C 180,E1 -23054.227,E2 -23054.227} C_VEL
LIN {X 0,Y 171.548,Z 374.114,A -85,B 0,C 180,E1 -23059.563,E2 -23059.563} C_VEL
LIN {X 0,Y 171.472,Z 374.121,A -85,B 0,C 180,E1 -23065.616,E2 -23065.616} C_VEL
LIN {X 0,Y 171.443,Z 374.128,A -85,B 0,C 180,E1 -23070.586,E2 -23070.586} C_VEL
LIN {X 0,Y 171.418,Z 374.127,A -85,B 0,C 180,E1 -23075.029,E2 -23075.029} C_VEL
LIN {X 0,Y 171.819,Z 374.144,A -85,B 0,C 180,E1 -23081.561,E2 -23081.561} C_VEL
LIN {X 0,Y 173.68,Z 382.527,A -85,B 0,C 180,E1 -23088.35,E2 -23088.35} C_VEL
LIN {X 0,Y 174.24,Z 384.66,A -85,B 0,C 180,E1 -23090.03,E2 -23090.03} C_VEL
LIN {X 0,Y 174.465,Z 386.519,A -85,B 0,C 180,E1 -23091.471,E2 -23091.471} C_VEL
LIN {X 0,Y 173.285,Z 391.536,A -85,B 0,C 180,E1 -23095.402,E2 -23095.402} C_VEL
LIN {X 0,Y 171.412,Z 401.284,A -85,B 0,C 180,E1 -23103.191,E2 -23103.191} C_VEL
LIN {X 0,Y 171.095,Z 404.184,A -85,B 0,C 180,E1 -23105.568,E2 -23105.568} C_VEL
LIN {X 0,Y 170.534,Z 416.473,A -85,B 0,C 180,E1 -23106.951,E2 -23106.951} C_VEL
LIN {X 0,Y 170.711,Z 429.75,A -85,B 0,C 180,E1 -23108.886,E2 -23108.886} C_VEL
LIN {X 0,Y 171.402,Z 442.176,A -85,B 0,C 180,E1 -23111.161,E2 -23111.161} C_VEL
LIN {X 0,Y 172.436,Z 453.721,A -85,B 0,C 180,E1 -23113.727,E2 -23113.727} C_VEL
LIN {X 0,Y 173.406,Z 462.076,A -85,B 0,C 180,E1 -23115.926,E2 -23115.926} C_VEL
LIN {X 0,Y 173.254,Z 471.086,A -85,B 0,C 180,E1 -23118.89,E2 -23118.89} C_VEL
LIN {X 0,Y 173.367,Z 479.773,A -85,B 0,C 180,E1 -23122.429,E2 -23122.429} C_VEL
LIN {X 0,Y 173.954,Z 486.729,A -85,B 0,C 180,E1 -23125.945,E2 -23125.945} C_VEL
LIN {X 0,Y 174.624,Z 491.336,A -85,B 0,C 180,E1 -23128.847,E2 -23128.847} C_VEL
LIN {X 0,Y 174.836,Z 492.894,A -85,B 0,C 180,E1 -23130,E2 -23130} C_VEL
LIN {X 0,Y 174.078,Z 495.082,A -85,B 0,C 180,E1 -23132.314,E2 -23132.314} C_VEL
LIN {X 0,Y 172.13,Z 497.911,A -85,B 0,C 180,E1 -23137.036,E2 -23137.036} C_VEL
LIN {X 0,Y 171.331,Z 499.408,A -85,B 0,C 180,E1 -23141.835,E2 -23141.835} C_VEL
LIN {X 0,Y 172.001,Z 499.767,A -85,B 0,C 180,E1 -23146.62,E2 -23146.62} C_VEL
LIN {X 0,Y 174.249,Z 499.089,A -85,B 0,C 180,E1 -23151.284,E2 -23151.284} C_VEL
LIN {X 0,Y 178.18,Z 497.412,A -85,B 0,C 180,E1 -23155.714,E2 -23155.714} C_VEL
LIN {X 0,Y 183.537,Z 494.701,A -85,B 0,C 180,E1 -23159.854,E2 -23159.854} C_VEL
LIN {X 0,Y 190.263,Z 490.624,A -85,B 0,C 180,E1 -23164.008,E2 -23164.008} C_VEL
LIN {X 0,Y 192.511,Z 488.882,A -85,B 0,C 180,E1 -23165.561,E2 -23165.561} C_VEL
LIN {X 0,Y 194.91,Z 485.94,A -85,B 0,C 180,E1 -23168.273,E2 -23168.273} C_VEL
LIN {X 0,Y 196.832,Z 483.446,A -85,B 0,C 180,E1 -23170.423,E2 -23170.423} C_VEL
LIN {X 0,Y 199.876,Z 480.706,A -85,B 0,C 180,E1 -23172.391,E2 -23172.391} C_VEL
LIN {X 0,Y 206.422,Z 475.567,A -85,B 0,C 180,E1 -23175.642,E2 -23175.642} C_VEL
LIN {X 0,Y 211.524,Z 471.366,A -85,B 0,C 180,E1 -23178.355,E2 -23178.355} C_VEL
LIN {X 0,Y 212.746,Z 470.123,A -85,B 0,C 180,E1 -23179.447,E2 -23179.447} C_VEL
LIN {X 0,Y 213.19,Z 468.511,A -85,B 0,C 180,E1 -23182.297,E2 -23182.297} C_VEL
LIN {X 0,Y 211.759,Z 468.781,A -85,B 0,C 180,E1 -23183.316,E2 -23183.316} C_VEL
LIN {X 0,Y 202.682,Z 471.386,A -85,B 0,C 180,E1 -23186.303,E2 -23186.303} C_VEL
LIN {X 0,Y 194.381,Z 472.741,A -85,B 0,C 180,E1 -23189.59,E2 -23189.59} C_VEL
LIN {X 0,Y 186.931,Z 472.847,A -85,B 0,C 180,E1 -23193.181,E2 -23193.181} C_VEL
LIN {X 0,Y 180.355,Z 471.68,A -85,B 0,C 180,E1 -23197.065,E2 -23197.065} C_VEL
LIN {X 0,Y 174.867,Z 469.223,A -85,B 0,C 180,E1 -23201.244,E2 -23201.244} C_VEL
LIN {X 0,Y 170.54,Z 465.471,A -85,B 0,C 180,E1 -23205.684,E2 -23205.684} C_VEL
LIN {X 0,Y 167.244,Z 460.299,A -85,B 0,C 180,E1 -23210.323,E2 -23210.323} C_VEL
LIN {X 0,Y 165.169,Z 453.629,A -85,B 0,C 180,E1 -23215.118,E2 -23215.118} C_VEL
LIN {X 0,Y 164.359,Z 446.401,A -85,B 0,C 180,E1 -23219.387,E2 -23219.387} C_VEL
LIN {X 0,Y 164.063,Z 437.549,A -85,B 0,C 180,E1 -23223.684,E2 -23223.684} C_VEL
LIN {X 0,Y 164.457,Z 428.497,A -85,B 0,C 180,E1 -23227.365,E2 -23227.365} C_VEL
LIN {X 0,Y 165.131,Z 419.618,A -85,B 0,C 180,E1 -23230.421,E2 -23230.421} C_VEL
LIN {X 0,Y 166.255,Z 408.267,A -85,B 0,C 180,E1 -23233.684,E2 -23233.684} C_VEL
LIN {X 0,Y 167.446,Z 395.149,A -85,B 0,C 180,E1 -23236.771,E2 -23236.771} C_VEL
LIN {X 0,Y 167.915,Z 390.755,A -85,B 0,C 180,E1 -23237.664,E2 -23237.664} C_VEL
LIN {X 0,Y 165.285,Z 378.147,A -85,B 0,C 180,E1 -23239.886,E2 -23239.886} C_VEL
LIN {X 0,Y 164.732,Z 374.964,A -85,B 0,C 180,E1 -23240.439,E2 -23240.439} C_VEL
LIN {X 0,Y 164.395,Z 375.001,A -85,B 0,C 180,E1 -23246.134,E2 -23246.134} C_VEL
LIN {X 0,Y 164.39,Z 375.007,A -85,B 0,C 180,E1 -23251.236,E2 -23251.236} C_VEL
LIN {X 0,Y 164.348,Z 375.012,A -85,B 0,C 180,E1 -23256.775,E2 -23256.775} C_VEL
LIN {X 0,Y 164.336,Z 375.013,A -85,B 0,C 180,E1 -23259.902,E2 -23259.902} C_VEL
LIN {X 0,Y 164.307,Z 375.014,A -85,B 0,C 180,E1 -23263.352,E2 -23263.352} C_VEL
LIN {X 0,Y 164.292,Z 375.021,A -85,B 0,C 180,E1 -23266.808,E2 -23266.808} C_VEL
LIN {X 0,Y 164.306,Z 375.016,A -85,B 0,C 180,E1 -23270.347,E2 -23270.347} C_VEL
LIN {X 0,Y 164.344,Z 375.013,A -85,B 0,C 180,E1 -23274.342,E2 -23274.342} C_VEL
LIN {X 0,Y 164.391,Z 375.002,A -85,B 0,C 180,E1 -23279.135,E2 -23279.135} C_VEL
LIN {X 0,Y 164.419,Z 375.004,A -85,B 0,C 180,E1 -23284.694,E2 -23284.694} C_VEL
LIN {X 0,Y 164.52,Z 374.988,A -85,B 0,C 180,E1 -23290.017,E2 -23290.017} C_VEL
LIN {X 0,Y 164.531,Z 374.987,A -85,B 0,C 180,E1 -23295.15,E2 -23295.15} C_VEL
LIN {X 0,Y 164.769,Z 374.961,A -85,B 0,C 180,E1 -23300.177,E2 -23300.177} C_VEL
LIN {X 0,Y 164.832,Z 374.951,A -85,B 0,C 180,E1 -23302.651,E2 -23302.651} C_VEL
LIN {X 0,Y 165.049,Z 374.923,A -85,B 0,C 180,E1 -23307.56,E2 -23307.56} C_VEL
LIN {X 0,Y 165.296,Z 374.896,A -85,B 0,C 180,E1 -23310,E2 -23310} C_VEL
LIN {X 0,Y 164.767,Z 374.955,A -85,B 0,C 180,E1 -23314.894,E2 -23314.894} C_VEL
LIN {X 0,Y 164.832,Z 374.951,A -85,B 0,C 180,E1 -23317.349,E2 -23317.349} C_VEL
LIN {X 0,Y 164.615,Z 374.974,A -85,B 0,C 180,E1 -23322.326,E2 -23322.326} C_VEL
LIN {X 0,Y 164.499,Z 374.995,A -85,B 0,C 180,E1 -23327.402,E2 -23327.402} C_VEL
LIN {X 0,Y 164.476,Z 374.993,A -85,B 0,C 180,E1 -23329.989,E2 -23329.989} C_VEL
LIN {X 0,Y 164.394,Z 375.006,A -85,B 0,C 180,E1 -23336.135,E2 -23336.135} C_VEL
LIN {X 0,Y 164.377,Z 375.005,A -85,B 0,C 180,E1 -23341.229,E2 -23341.229} C_VEL
LIN {X 0,Y 164.352,Z 375.01,A -85,B 0,C 180,E1 -23346.775,E2 -23346.775} C_VEL
LIN {X 0,Y 164.373,Z 375.007,A -85,B 0,C 180,E1 -23349.893,E2 -23349.893} C_VEL
LIN {X 0,Y 164.341,Z 375.015,A -85,B 0,C 180,E1 -23353.365,E2 -23353.365} C_VEL
LIN {X 0,Y 164.322,Z 375.012,A -85,B 0,C 180,E1 -23356.819,E2 -23356.819} C_VEL
LIN {X 0,Y 164.3,Z 375.017,A -85,B 0,C 180,E1 -23360.351,E2 -23360.351} C_VEL
LIN {X 0,Y 164.331,Z 375.009,A -85,B 0,C 180,E1 -23366.223,E2 -23366.223} C_VEL
LIN {X 0,Y 164.407,Z 375.007,A -85,B 0,C 180,E1 -23369.139,E2 -23369.139} C_VEL
LIN {X 0,Y 164.419,Z 374.999,A -85,B 0,C 180,E1 -23374.695,E2 -23374.695} C_VEL
LIN {X 0,Y 164.488,Z 374.994,A -85,B 0,C 180,E1 -23380.05,E2 -23380.05} C_VEL
LIN {X 0,Y 164.562,Z 374.986,A -85,B 0,C 180,E1 -23385.153,E2 -23385.153} C_VEL
LIN {X 0,Y 164.856,Z 374.947,A -85,B 0,C 180,E1 -23390.182,E2 -23390.182} C_VEL
LIN {X 0,Y 164.866,Z 374.945,A -85,B 0,C 180,E1 -23392.653,E2 -23392.653} C_VEL
LIN {X 0,Y 165.054,Z 374.923,A -85,B 0,C 180,E1 -23397.56,E2 -23397.56} C_VEL
LIN {X 0,Y 165.299,Z 374.889,A -85,B 0,C 180,E1 -23400,E2 -23400} C_VEL
LIN {X 0,Y 164.768,Z 374.96,A -85,B 0,C 180,E1 -23404.894,E2 -23404.894} C_VEL
LIN {X 0,Y 164.833,Z 374.948,A -85,B 0,C 180,E1 -23407.349,E2 -23407.349} C_VEL
LIN {X 0,Y 164.706,Z 374.967,A -85,B 0,C 180,E1 -23411.062,E2 -23411.062} C_VEL
LIN {X 0,Y 164.487,Z 374.989,A -85,B 0,C 180,E1 -23417.403,E2 -23417.403} C_VEL
LIN {X 0,Y 164.477,Z 374.996,A -85,B 0,C 180,E1 -23419.989,E2 -23419.989} C_VEL
LIN {X 0,Y 164.396,Z 375.003,A -85,B 0,C 180,E1 -23426.134,E2 -23426.134} C_VEL
LIN {X 0,Y 164.377,Z 375.008,A -85,B 0,C 180,E1 -23431.227,E2 -23431.227} C_VEL
LIN {X 0,Y 164.384,Z 375.007,A -85,B 0,C 180,E1 -23436.767,E2 -23436.767} C_VEL
LIN {X 0,Y 164.829,Z 375.093,A -85,B 0,C 180,E1 -23441.982,E2 -23441.982} C_VEL
LIN {X 0,Y 166.869,Z 383.801,A -85,B 0,C 180,E1 -23449.298,E2 -23449.298} C_VEL
LIN {X 0,Y 167.272,Z 385.796,A -85,B 0,C 180,E1 -23450.932,E2 -23450.932} C_VEL
LIN {X 0,Y 166.674,Z 389.299,A -85,B 0,C 180,E1 -23453.819,E2 -23453.819} C_VEL
LIN {X 0,Y 165.061,Z 395.842,A -85,B 0,C 180,E1 -23459.273,E2 -23459.273} C_VEL
LIN {X 0,Y 164.059,Z 403.133,A -85,B 0,C 180,E1 -23465.481,E2 -23465.481} C_VEL
LIN {X 0,Y 163.477,Z 418.394,A -85,B 0,C 180,E1 -23467.404,E2 -23467.404} C_VEL
LIN {X 0,Y 163.794,Z 431.902,A -85,B 0,C 180,E1 -23469.597,E2 -23469.597} C_VEL
LIN {X 0,Y 164.599,Z 443.873,A -85,B 0,C 180,E1 -23471.994,E2 -23471.994} C_VEL
LIN {X 0,Y 165.849,Z 455.959,A -85,B 0,C 180,E1 -23474.956,E2 -23474.956} C_VEL
LIN {X 0,Y 166.592,Z 462.777,A -85,B 0,C 180,E1 -23476.927,E2 -23476.927} C_VEL
LIN {X 0,Y 166.482,Z 471.994,A -85,B 0,C 180,E1 -23480.278,E2 -23480.278} C_VEL
LIN {X 0,Y 166.802,Z 480.243,A -85,B 0,C 180,E1 -23483.953,E2 -23483.953} C_VEL
LIN {X 0,Y 167.546,Z 486.752,A -85,B 0,C 180,E1 -23487.596,E2 -23487.596} C_VEL
LIN {X 0,Y 168.109,Z 490.226,A -85,B 0,C 180,E1 -23490,E2 -23490} C_VEL
LIN {X 0,Y 167.912,Z 491.564,A -85,B 0,C 180,E1 -23491.199,E2 -23491.199} C_VEL
LIN {X 0,Y 166.225,Z 494.32,A -85,B 0,C 180,E1 -23494.851,E2 -23494.851} C_VEL
LIN {X 0,Y 164.766,Z 496.691,A -85,B 0,C 180,E1 -23499.824,E2 -23499.824} C_VEL
LIN {X 0,Y 164.764,Z 497.863,A -85,B 0,C 180,E1 -23504.829,E2 -23504.829} C_VEL
LIN {X 0,Y 166.295,Z 497.968,A -85,B 0,C 180,E1 -23509.761,E2 -23509.761} C_VEL
LIN {X 0,Y 169.595,Z 497.116,A -85,B 0,C 180,E1 -23514.481,E2 -23514.481} C_VEL
LIN {X 0,Y 174.441,Z 495.274,A -85,B 0,C 180,E1 -23518.912,E2 -23518.912} C_VEL
LIN {X 0,Y 180.602,Z 492.428,A -85,B 0,C 180,E1 -23523.011,E2 -23523.011} C_VEL
LIN {X 0,Y 187.556,Z 488.593,A -85,B 0,C 180,E1 -23526.837,E2 -23526.837} C_VEL
LIN {X 0,Y 195.438,Z 483.84,A -85,B 0,C 180,E1 -23530.337,E2 -23530.337} C_VEL
LIN {X 0,Y 199.876,Z 480.706,A -85,B 0,C 180,E1 -23532.391,E2 -23532.391} C_VEL
LIN {X 0,Y 202.302,Z 478.664,A -85,B 0,C 180,E1 -23533.824,E2 -23533.824} C_VEL
LIN {X 0,Y 204.286,Z 476.32,A -85,B 0,C 180,E1 -23535.894,E2 -23535.894} C_VEL
LIN {X 0,Y 205.584,Z 473.913,A -85,B 0,C 180,E1 -23538.622,E2 -23538.622} C_VEL
LIN {X 0,Y 206.351,Z 472.304,A -85,B 0,C 180,E1 -23540.836,E2 -23540.836} C_VEL
LIN {X 0,Y 206.609,Z 471.866,A -85,B 0,C 180,E1 -23541.478,E2 -23541.478} C_VEL
LIN {X 0,Y 206.4,Z 471.613,A -85,B 0,C 180,E1 -23542.199,E2 -23542.199} C_VEL
LIN {X 0,Y 197.108,Z 473.682,A -85,B 0,C 180,E1 -23545.215,E2 -23545.215} C_VEL
LIN {X 0,Y 188.486,Z 474.57,A -85,B 0,C 180,E1 -23548.532,E2 -23548.532} C_VEL
LIN {X 0,Y 180.76,Z 474.237,A -85,B 0,C 180,E1 -23552.188,E2 -23552.188} C_VEL
LIN {X 0,Y 173.913,Z 472.681,A -85,B 0,C 180,E1 -23556.164,E2 -23556.164} C_VEL
LIN {X 0,Y 168.205,Z 469.802,A -85,B 0,C 180,E1 -23560.472,E2 -23560.472} C_VEL
LIN {X 0,Y 163.672,Z 465.632,A -85,B 0,C 180,E1 -23565.07,E2 -23565.07} C_VEL
LIN {X 0,Y 160.255,Z 460.106,A -85,B 0,C 180,E1 -23569.896,E2 -23569.896} C_VEL
LIN {X 0,Y 158.117,Z 453.001,A -85,B 0,C 180,E1 -23574.899,E2 -23574.899} C_VEL
LIN {X 0,Y 157.319,Z 445.402,A -85,B 0,C 180,E1 -23579.36,E2 -23579.36} C_VEL
LIN {X 0,Y 157.031,Z 436.149,A -85,B 0,C 180,E1 -23583.849,E2 -23583.849} C_VEL
LIN {X 0,Y 157.672,Z 424.93,A -85,B 0,C 180,E1 -23588.329,E2 -23588.329} C_VEL
LIN {X 0,Y 158.637,Z 413.217,A -85,B 0,C 180,E1 -23592.122,E2 -23592.122} C_VEL
LIN {X 0,Y 159.749,Z 401.28,A -85,B 0,C 180,E1 -23595.305,E2 -23595.305} C_VEL
LIN {X 0,Y 160.745,Z 391.413,A -85,B 0,C 180,E1 -23597.492,E2 -23597.492} C_VEL
LIN {X 0,Y 158.207,Z 378.784,A -85,B 0,C 180,E1 -23599.799,E2 -23599.799} C_VEL
LIN {X 0,Y 157.699,Z 375.84,A -85,B 0,C 180,E1 -23600.287,E2 -23600.287} C_VEL
LIN {X 0,Y 157.316,Z 375.884,A -85,B 0,C 180,E1 -23606.685,E2 -23606.685} C_VEL
LIN {X 0,Y 157.284,Z 375.891,A -85,B 0,C 180,E1 -23612.425,E2 -23612.425} C_VEL
LIN {X 0,Y 157.323,Z 375.886,A -85,B 0,C 180,E1 -23616.476,E2 -23616.476} C_VEL
LIN {X 0,Y 157.241,Z 375.894,A -85,B 0,C 180,E1 -23622.1,E2 -23622.1} C_VEL
LIN {X 0,Y 157.213,Z 375.901,A -85,B 0,C 180,E1 -23627.89,E2 -23627.89} C_VEL
LIN {X 0,Y 157.283,Z 375.891,A -85,B 0,C 180,E1 -23633.543,E2 -23633.543} C_VEL
LIN {X 0,Y 157.295,Z 375.89,A -85,B 0,C 180,E1 -23638.094,E2 -23638.094} C_VEL
LIN {X 0,Y 157.323,Z 375.887,A -85,B 0,C 180,E1 -23643.466,E2 -23643.466} C_VEL
LIN {X 0,Y 157.447,Z 375.868,A -85,B 0,C 180,E1 -23649.616,E2 -23649.616} C_VEL
LIN {X 0,Y 157.464,Z 375.869,A -85,B 0,C 180,E1 -23654.467,E2 -23654.467} C_VEL
LIN {X 0,Y 157.69,Z 375.841,A -85,B 0,C 180,E1 -23659.731,E2 -23659.731} C_VEL
LIN {X 0,Y 157.769,Z 375.832,A -85,B 0,C 180,E1 -23662.32,E2 -23662.32} C_VEL
LIN {X 0,Y 158.258,Z 375.773,A -85,B 0,C 180,E1 -23670,E2 -23670} C_VEL
LIN {X 0,Y 157.769,Z 375.832,A -85,B 0,C 180,E1 -23677.68,E2 -23677.68} C_VEL
LIN {X 0,Y 157.638,Z 375.847,A -85,B 0,C 180,E1 -23681.238,E2 -23681.238} C_VEL
LIN {X 0,Y 157.462,Z 375.87,A -85,B 0,C 180,E1 -23685.534,E2 -23685.534} C_VEL
LIN {X 0,Y 157.372,Z 375.877,A -85,B 0,C 180,E1 -23690.933,E2 -23690.933} C_VEL
LIN {X 0,Y 157.316,Z 375.888,A -85,B 0,C 180,E1 -23696.686,E2 -23696.686} C_VEL
LIN {X 0,Y 157.279,Z 375.891,A -85,B 0,C 180,E1 -23702.427,E2 -23702.427} C_VEL
LIN {X 0,Y 157.326,Z 375.885,A -85,B 0,C 180,E1 -23706.478,E2 -23706.478} C_VEL
LIN {X 0,Y 157.272,Z 375.893,A -85,B 0,C 180,E1 -23712.091,E2 -23712.091} C_VEL
LIN {X 0,Y 157.231,Z 375.895,A -85,B 0,C 180,E1 -23717.896,E2 -23717.896} C_VEL
LIN {X 0,Y 157.27,Z 375.892,A -85,B 0,C 180,E1 -23723.551,E2 -23723.551} C_VEL
LIN {X 0,Y 157.303,Z 375.888,A -85,B 0,C 180,E1 -23728.092,E2 -23728.092} C_VEL
LIN {X 0,Y 157.324,Z 375.882,A -85,B 0,C 180,E1 -23733.467,E2 -23733.467} C_VEL
LIN {X 0,Y 157.398,Z 375.877,A -85,B 0,C 180,E1 -23739.666,E2 -23739.666} C_VEL
LIN {X 0,Y 157.489,Z 375.864,A -85,B 0,C 180,E1 -23744.47,E2 -23744.47} C_VEL
LIN {X 0,Y 157.775,Z 375.829,A -85,B 0,C 180,E1 -23749.737,E2 -23749.737} C_VEL
LIN {X 0,Y 157.828,Z 375.82,A -85,B 0,C 180,E1 -23752.323,E2 -23752.323} C_VEL
LIN {X 0,Y 158.261,Z 375.766,A -85,B 0,C 180,E1 -23760,E2 -23760} C_VEL
LIN {X 0,Y 157.77,Z 375.828,A -85,B 0,C 180,E1 -23767.68,E2 -23767.68} C_VEL
LIN {X 0,Y 157.64,Z 375.847,A -85,B 0,C 180,E1 -23771.238,E2 -23771.238} C_VEL
LIN {X 0,Y 157.457,Z 375.869,A -85,B 0,C 180,E1 -23775.534,E2 -23775.534} C_VEL
LIN {X 0,Y 157.373,Z 375.881,A -85,B 0,C 180,E1 -23780.933,E2 -23780.933} C_VEL
LIN {X 0,Y 157.317,Z 375.885,A -85,B 0,C 180,E1 -23786.685,E2 -23786.685} C_VEL
LIN {X 0,Y 157.281,Z 375.89,A -85,B 0,C 180,E1 -23792.427,E2 -23792.427} C_VEL
LIN {X 0,Y 157.432,Z 375.874,A -85,B 0,C 180,E1 -23798.681,E2 -23798.681} C_VEL
LIN {X 0,Y 157.799,Z 375.9,A -85,B 0,C 180,E1 -23802.349,E2 -23802.349} C_VEL
LIN {X 0,Y 159.75,Z 383.87,A -85,B 0,C 180,E1 -23809.365,E2 -23809.365} C_VEL
LIN {X 0,Y 160.073,Z 387.036,A -85,B 0,C 180,E1 -23812.071,E2 -23812.071} C_VEL
LIN {X 0,Y 158.458,Z 393.171,A -85,B 0,C 180,E1 -23817.427,E2 -23817.427} C_VEL
LIN {X 0,Y 157.268,Z 399.894,A -85,B 0,C 180,E1 -23823.456,E2 -23823.456} C_VEL
LIN {X 0,Y 157.045,Z 402.247,A -85,B 0,C 180,E1 -23825.546,E2 -23825.546} C_VEL
LIN {X 0,Y 156.447,Z 414.057,A -85,B 0,C 180,E1 -23827.029,E2 -23827.029} C_VEL
LIN {X 0,Y 156.586,Z 427.315,A -85,B 0,C 180,E1 -23829.157,E2 -23829.157} C_VEL
LIN {X 0,Y 157.37,Z 440.366,A -85,B 0,C 180,E1 -23831.783,E2 -23831.783} C_VEL
LIN {X 0,Y 158.495,Z 451.766,A -85,B 0,C 180,E1 -23834.57,E2 -23834.57} C_VEL
LIN {X 0,Y 159.737,Z 461.127,A -85,B 0,C 180,E1 -23837.292,E2 -23837.292} C_VEL
LIN {X 0,Y 159.737,Z 471.217,A -85,B 0,C 180,E1 -23841.141,E2 -23841.141} C_VEL
LIN {X 0,Y 160.218,Z 479.309,A -85,B 0,C 180,E1 -23844.967,E2 -23844.967} C_VEL
LIN {X 0,Y 161.077,Z 485.674,A -85,B 0,C 180,E1 -23848.75,E2 -23848.75} C_VEL
LIN {X 0,Y 161.362,Z 487.444,A -85,B 0,C 180,E1 -23850,E2 -23850} C_VEL
LIN {X 0,Y 161.339,Z 488.9,A -85,B 0,C 180,E1 -23851.248,E2 -23851.248} C_VEL
LIN {X 0,Y 159.534,Z 491.83,A -85,B 0,C 180,E1 -23855.055,E2 -23855.055} C_VEL
LIN {X 0,Y 158.035,Z 494.428,A -85,B 0,C 180,E1 -23860.246,E2 -23860.246} C_VEL
LIN {X 0,Y 158.06,Z 495.853,A -85,B 0,C 180,E1 -23865.473,E2 -23865.473} C_VEL
LIN {X 0,Y 159.747,Z 496.255,A -85,B 0,C 180,E1 -23870.607,E2 -23870.607} C_VEL
LIN {X 0,Y 163.219,Z 495.729,A -85,B 0,C 180,E1 -23875.505,E2 -23875.505} C_VEL
LIN {X 0,Y 168.309,Z 494.248,A -85,B 0,C 180,E1 -23880.071,E2 -23880.071} C_VEL
LIN {X 0,Y 174.669,Z 491.782,A -85,B 0,C 180,E1 -23884.285,E2 -23884.285} C_VEL
LIN {X 0,Y 183.93,Z 487.389,A -85,B 0,C 180,E1 -23889.085,E2 -23889.085} C_VEL
LIN {X 0,Y 190.046,Z 484.065,A -85,B 0,C 180,E1 -23891.732,E2 -23891.732} C_VEL
LIN {X 0,Y 195.683,Z 480.514,A -85,B 0,C 180,E1 -23894.311,E2 -23894.311} C_VEL
LIN {X 0,Y 201.432,Z 476.498,A -85,B 0,C 180,E1 -23897.113,E2 -23897.113} C_VEL
LIN {X 0,Y 205.021,Z 473.909,A -85,B 0,C 180,E1 -23898.951,E2 -23898.951} C_VEL
LIN {X 0,Y 205.921,Z 473.163,A -85,B 0,C 180,E1 -23899.574,E2 -23899.574} C_VEL
LIN {X 0,Y 206.351,Z 472.304,A -85,B 0,C 180,E1 -23900.836,E2 -23900.836} C_VEL
LIN {X 0,Y 205.852,Z 472.197,A -85,B 0,C 180,E1 -23901.466,E2 -23901.466} C_VEL
LIN {X 0,Y 203.959,Z 472.615,A -85,B 0,C 180,E1 -23902.133,E2 -23902.133} C_VEL
LIN {X 0,Y 200.205,Z 473.698,A -85,B 0,C 180,E1 -23902.832,E2 -23902.832} C_VEL
LIN {X 0,Y 193.442,Z 475.453,A -85,B 0,C 180,E1 -23903.776,E2 -23903.776} C_VEL
LIN {X 0,Y 189.947,Z 475.997,A -85,B 0,C 180,E1 -23904.618,E2 -23904.618} C_VEL
LIN {X 0,Y 182.64,Z 476.275,A -85,B 0,C 180,E1 -23907.403,E2 -23907.403} C_VEL
LIN {X 0,Y 174.606,Z 475.492,A -85,B 0,C 180,E1 -23911.117,E2 -23911.117} C_VEL
LIN {X 0,Y 167.5,Z 473.496,A -85,B 0,C 180,E1 -23915.191,E2 -23915.191} C_VEL
LIN {X 0,Y 161.557,Z 470.244,A -85,B 0,C 180,E1 -23919.634,E2 -23919.634} C_VEL
LIN {X 0,Y 156.821,Z 465.663,A -85,B 0,C 180,E1 -23924.401,E2 -23924.401} C_VEL
LIN {X 0,Y 153.278,Z 459.707,A -85,B 0,C 180,E1 -23929.431,E2 -23929.431} C_VEL
LIN {X 0,Y 151.083,Z 452.222,A -85,B 0,C 180,E1 -23934.661,E2 -23934.661} C_VEL
LIN {X 0,Y 150.275,Z 444.209,A -85,B 0,C 180,E1 -23939.33,E2 -23939.33} C_VEL
LIN {X 0,Y 150.024,Z 434.526,A -85,B 0,C 180,E1 -23944.029,E2 -23944.029} C_VEL
LIN {X 0,Y 150.733,Z 422.738,A -85,B 0,C 180,E1 -23948.715,E2 -23948.715} C_VEL
LIN {X 0,Y 151.795,Z 410.417,A -85,B 0,C 180,E1 -23952.676,E2 -23952.676} C_VEL
LIN {X 0,Y 152.984,Z 397.736,A -85,B 0,C 180,E1 -23956,E2 -23956} C_VEL
LIN {X 0,Y 153.587,Z 391.873,A -85,B 0,C 180,E1 -23957.303,E2 -23957.303} C_VEL
LIN {X 0,Y 152.259,Z 384.905,A -85,B 0,C 180,E1 -23958.676,E2 -23958.676} C_VEL
LIN {X 0,Y 150.66,Z 376.717,A -85,B 0,C 180,E1 -23960.165,E2 -23960.165} C_VEL
LIN {X 0,Y 150.226,Z 376.77,A -85,B 0,C 180,E1 -23967.893,E2 -23967.893} C_VEL
LIN {X 0,Y 150.224,Z 376.771,A -85,B 0,C 180,E1 -23972.637,E2 -23972.637} C_VEL
LIN {X 0,Y 150.226,Z 376.772,A -85,B 0,C 180,E1 -23977.457,E2 -23977.457} C_VEL
LIN {X 0,Y 150.184,Z 376.773,A -85,B 0,C 180,E1 -23981.519,E2 -23981.519} C_VEL
LIN {X 0,Y 150.154,Z 376.78,A -85,B 0,C 180,E1 -23985.406,E2 -23985.406} C_VEL
LIN {X 0,Y 150.157,Z 376.779,A -85,B 0,C 180,E1 -23989.06,E2 -23989.06} C_VEL
LIN {X 0,Y 150.216,Z 376.77,A -85,B 0,C 180,E1 -23992.689,E2 -23992.689} C_VEL
LIN {X 0,Y 150.219,Z 376.771,A -85,B 0,C 180,E1 -23997.365,E2 -23997.365} C_VEL
LIN {X 0,Y 150.245,Z 376.77,A -85,B 0,C 180,E1 -24002.717,E2 -24002.717} C_VEL
LIN {X 0,Y 150.39,Z 376.746,A -85,B 0,C 180,E1 -24009.169,E2 -24009.169} C_VEL
LIN {X 0,Y 150.376,Z 376.753,A -85,B 0,C 180,E1 -24013.715,E2 -24013.715} C_VEL
LIN {X 0,Y 150.612,Z 376.721,A -85,B 0,C 180,E1 -24019.243,E2 -24019.243} C_VEL
LIN {X 0,Y 150.706,Z 376.713,A -85,B 0,C 180,E1 -24021.958,E2 -24021.958} C_VEL
LIN {X 0,Y 151.219,Z 376.65,A -85,B 0,C 180,E1 -24030,E2 -24030} C_VEL
LIN {X 0,Y 150.706,Z 376.713,A -85,B 0,C 180,E1 -24038.042,E2 -24038.042} C_VEL
LIN {X 0,Y 150.578,Z 376.726,A -85,B 0,C 180,E1 -24041.439,E2 -24041.439} C_VEL
LIN {X 0,Y 150.371,Z 376.754,A -85,B 0,C 180,E1 -24046.286,E2 -24046.286} C_VEL
LIN {X 0,Y 150.353,Z 376.751,A -85,B 0,C 180,E1 -24050.794,E2 -24050.794} C_VEL
LIN {X 0,Y 150.245,Z 376.77,A -85,B 0,C 180,E1 -24057.283,E2 -24057.283} C_VEL
LIN {X 0,Y 150.22,Z 376.771,A -85,B 0,C 180,E1 -24062.635,E2 -24062.635} C_VEL
LIN {X 0,Y 150.237,Z 376.766,A -85,B 0,C 180,E1 -24067.455,E2 -24067.455} C_VEL
LIN {X 0,Y 150.218,Z 376.774,A -85,B 0,C 180,E1 -24071.534,E2 -24071.534} C_VEL
LIN {X 0,Y 150.168,Z 376.776,A -85,B 0,C 180,E1 -24075.412,E2 -24075.412} C_VEL
LIN {X 0,Y 150.164,Z 376.777,A -85,B 0,C 180,E1 -24079.063,E2 -24079.063} C_VEL
LIN {X 0,Y 150.184,Z 376.777,A -85,B 0,C 180,E1 -24082.706,E2 -24082.706} C_VEL
LIN {X 0,Y 150.222,Z 376.771,A -85,B 0,C 180,E1 -24087.365,E2 -24087.365} C_VEL
LIN {X 0,Y 150.247,Z 376.767,A -85,B 0,C 180,E1 -24092.718,E2 -24092.718} C_VEL
LIN {X 0,Y 150.355,Z 376.756,A -85,B 0,C 180,E1 -24099.207,E2 -24099.207} C_VEL
LIN {X 0,Y 150.394,Z 376.746,A -85,B 0,C 180,E1 -24103.717,E2 -24103.717} C_VEL
LIN {X 0,Y 150.692,Z 376.711,A -85,B 0,C 180,E1 -24109.249,E2 -24109.249} C_VEL
LIN {X 0,Y 150.766,Z 376.698,A -85,B 0,C 180,E1 -24111.962,E2 -24111.962} C_VEL
LIN {X 0,Y 151.222,Z 376.642,A -85,B 0,C 180,E1 -24120,E2 -24120} C_VEL
LIN {X 0,Y 150.707,Z 376.708,A -85,B 0,C 180,E1 -24128.043,E2 -24128.043} C_VEL
LIN {X 0,Y 150.58,Z 376.726,A -85,B 0,C 180,E1 -24131.438,E2 -24131.438} C_VEL
LIN {X 0,Y 150.365,Z 376.75,A -85,B 0,C 180,E1 -24136.287,E2 -24136.287} C_VEL
LIN {X 0,Y 150.354,Z 376.756,A -85,B 0,C 180,E1 -24140.793,E2 -24140.793} C_VEL
LIN {X 0,Y 150.247,Z 376.766,A -85,B 0,C 180,E1 -24147.282,E2 -24147.282} C_VEL
LIN {X 0,Y 150.223,Z 376.769,A -85,B 0,C 180,E1 -24152.636,E2 -24152.636} C_VEL
LIN {X 0,Y 150.314,Z 376.76,A -85,B 0,C 180,E1 -24157.433,E2 -24157.433} C_VEL
LIN {X 0,Y 150.779,Z 376.797,A -85,B 0,C 180,E1 -24162.897,E2 -24162.897} C_VEL
LIN {X 0,Y 152.749,Z 384.403,A -85,B 0,C 180,E1 -24169.898,E2 -24169.898} C_VEL
LIN {X 0,Y 152.889,Z 387.09,A -85,B 0,C 180,E1 -24172.336,E2 -24172.336} C_VEL
LIN {X 0,Y 151.248,Z 393.064,A -85,B 0,C 180,E1 -24177.859,E2 -24177.859} C_VEL
LIN {X 0,Y 150.055,Z 400.652,A -85,B 0,C 180,E1 -24185.069,E2 -24185.069} C_VEL
LIN {X 0,Y 149.996,Z 401.476,A -85,B 0,C 180,E1 -24185.612,E2 -24185.612} C_VEL
LIN {X 0,Y 149.384,Z 414.246,A -85,B 0,C 180,E1 -24187.344,E2 -24187.344} C_VEL
LIN {X 0,Y 149.622,Z 427.863,A -85,B 0,C 180,E1 -24189.704,E2 -24189.704} C_VEL
LIN {X 0,Y 150.581,Z 441.546,A -85,B 0,C 180,E1 -24192.69,E2 -24192.69} C_VEL
LIN {X 0,Y 152.088,Z 453.971,A -85,B 0,C 180,E1 -24196.03,E2 -24196.03} C_VEL
LIN {X 0,Y 152.939,Z 460.407,A -85,B 0,C 180,E1 -24198.065,E2 -24198.065} C_VEL
LIN {X 0,Y 153.062,Z 470.345,A -85,B 0,C 180,E1 -24202.082,E2 -24202.082} C_VEL
LIN {X 0,Y 153.705,Z 478.283,A -85,B 0,C 180,E1 -24206.067,E2 -24206.067} C_VEL
LIN {X 0,Y 154.66,Z 484.502,A -85,B 0,C 180,E1 -24210,E2 -24210} C_VEL
LIN {X 0,Y 154.672,Z 486.356,A -85,B 0,C 180,E1 -24211.529,E2 -24211.529} C_VEL
LIN {X 0,Y 152.905,Z 489.213,A -85,B 0,C 180,E1 -24215.274,E2 -24215.274} C_VEL
LIN {X 0,Y 151.352,Z 492.034,A -85,B 0,C 180,E1 -24220.704,E2 -24220.704} C_VEL
LIN {X 0,Y 151.443,Z 493.72,A -85,B 0,C 180,E1 -24226.167,E2 -24226.167} C_VEL
LIN {X 0,Y 153.272,Z 494.393,A -85,B 0,C 180,E1 -24231.52,E2 -24231.52} C_VEL
LIN {X 0,Y 156.94,Z 494.177,A -85,B 0,C 180,E1 -24236.604,E2 -24236.604} C_VEL
LIN {X 0,Y 162.252,Z 493.059,A -85,B 0,C 180,E1 -24241.318,E2 -24241.318} C_VEL
LIN {X 0,Y 168.853,Z 490.994,A -85,B 0,C 180,E1 -24245.641,E2 -24245.641} C_VEL
LIN {X 0,Y 176.396,Z 487.98,A -85,B 0,C 180,E1 -24249.604,E2 -24249.604} C_VEL
LIN {X 0,Y 184.769,Z 484.126,A -85,B 0,C 180,E1 -24253.209,E2 -24253.209} C_VEL
LIN {X 0,Y 190.782,Z 480.782,A -85,B 0,C 180,E1 -24255.918,E2 -24255.918} C_VEL
LIN {X 0,Y 196.527,Z 477.23,A -85,B 0,C 180,E1 -24258.676,E2 -24258.676} C_VEL
LIN {X 0,Y 198.337,Z 476.084,A -85,B 0,C 180,E1 -24259.576,E2 -24259.576} C_VEL
LIN {X 0,Y 199.631,Z 474.962,A -85,B 0,C 180,E1 -24260.761,E2 -24260.761} C_VEL
LIN {X 0,Y 198.665,Z 474.749,A -85,B 0,C 180,E1 -24261.792,E2 -24261.792} C_VEL
LIN {X 0,Y 189.947,Z 475.997,A -85,B 0,C 180,E1 -24264.618,E2 -24264.618} C_VEL
LIN {X 0,Y 185.684,Z 476.423,A -85,B 0,C 180,E1 -24265.864,E2 -24265.864} C_VEL
LIN {X 0,Y 177.631,Z 476.95,A -85,B 0,C 180,E1 -24267.684,E2 -24267.684} C_VEL
LIN {X 0,Y 169.863,Z 476.702,A -85,B 0,C 180,E1 -24269.686,E2 -24269.686} C_VEL
LIN {X 0,Y 166.127,Z 475.95,A -85,B 0,C 180,E1 -24271.215,E2 -24271.215} C_VEL
LIN {X 0,Y 161.122,Z 474.168,A -85,B 0,C 180,E1 -24274.138,E2 -24274.138} C_VEL
LIN {X 0,Y 154.924,Z 470.488,A -85,B 0,C 180,E1 -24278.72,E2 -24278.72} C_VEL
LIN {X 0,Y 149.995,Z 465.539,A -85,B 0,C 180,E1 -24283.672,E2 -24283.672} C_VEL
LIN {X 0,Y 146.32,Z 459.151,A -85,B 0,C 180,E1 -24288.923,E2 -24288.923} C_VEL
LIN {X 0,Y 144.072,Z 451.248,A -85,B 0,C 180,E1 -24294.401,E2 -24294.401} C_VEL
LIN {X 0,Y 143.227,Z 442.828,A -85,B 0,C 180,E1 -24299.297,E2 -24299.297} C_VEL
LIN {X 0,Y 143.031,Z 432.631,A -85,B 0,C 180,E1 -24304.226,E2 -24304.226} C_VEL
LIN {X 0,Y 143.669,Z 422.2,A -85,B 0,C 180,E1 -24308.438,E2 -24308.438} C_VEL
LIN {X 0,Y 144.728,Z 409.763,A -85,B 0,C 180,E1 -24312.56,E2 -24312.56} C_VEL
LIN {X 0,Y 145.942,Z 396.882,A -85,B 0,C 180,E1 -24316.003,E2 -24316.003} C_VEL
LIN {X 0,Y 146.425,Z 392.155,A -85,B 0,C 180,E1 -24317.096,E2 -24317.096} C_VEL
LIN {X 0,Y 145.875,Z 388.421,A -85,B 0,C 180,E1 -24317.886,E2 -24317.886} C_VEL
LIN {X 0,Y 143.661,Z 377.589,A -85,B 0,C 180,E1 -24319.932,E2 -24319.932} C_VEL
LIN {X 0,Y 143.193,Z 377.646,A -85,B 0,C 180,E1 -24327.938,E2 -24327.938} C_VEL
LIN {X 0,Y 143.173,Z 377.645,A -85,B 0,C 180,E1 -24333.437,E2 -24333.437} C_VEL
LIN {X 0,Y 143.098,Z 377.659,A -85,B 0,C 180,E1 -24339.677,E2 -24339.677} C_VEL
LIN {X 0,Y 143.098,Z 377.655,A -85,B 0,C 180,E1 -24343.439,E2 -24343.439} C_VEL
LIN {X 0,Y 143.075,Z 377.662,A -85,B 0,C 180,E1 -24347.46,E2 -24347.46} C_VEL
LIN {X 0,Y 143.107,Z 377.652,A -85,B 0,C 180,E1 -24351.791,E2 -24351.791} C_VEL
LIN {X 0,Y 143.186,Z 377.647,A -85,B 0,C 180,E1 -24357.322,E2 -24357.322} C_VEL
LIN {X 0,Y 143.163,Z 377.651,A -85,B 0,C 180,E1 -24363.78,E2 -24363.78} C_VEL
LIN {X 0,Y 143.341,Z 377.625,A -85,B 0,C 180,E1 -24369.927,E2 -24369.927} C_VEL
LIN {X 0,Y 143.365,Z 377.624,A -85,B 0,C 180,E1 -24375.812,E2 -24375.812} C_VEL
LIN {X 0,Y 143.538,Z 377.603,A -85,B 0,C 180,E1 -24378.706,E2 -24378.706} C_VEL
LIN {X 0,Y 143.627,Z 377.594,A -85,B 0,C 180,E1 -24381.559,E2 -24381.559} C_VEL
LIN {X 0,Y 144.177,Z 377.527,A -85,B 0,C 180,E1 -24390,E2 -24390} C_VEL
LIN {X 0,Y 143.627,Z 377.594,A -85,B 0,C 180,E1 -24398.442,E2 -24398.442} C_VEL
LIN {X 0,Y 143.506,Z 377.605,A -85,B 0,C 180,E1 -24401.632,E2 -24401.632} C_VEL
LIN {X 0,Y 143.309,Z 377.633,A -85,B 0,C 180,E1 -24407.113,E2 -24407.113} C_VEL
LIN {X 0,Y 143.278,Z 377.632,A -85,B 0,C 180,E1 -24411.256,E2 -24411.256} C_VEL
LIN {X 0,Y 143.191,Z 377.646,A -85,B 0,C 180,E1 -24417.938,E2 -24417.938} C_VEL
LIN {X 0,Y 143.171,Z 377.651,A -85,B 0,C 180,E1 -24423.437,E2 -24423.437} C_VEL
LIN {X 0,Y 143.122,Z 377.654,A -85,B 0,C 180,E1 -24429.671,E2 -24429.671} C_VEL
LIN {X 0,Y 143.119,Z 377.658,A -85,B 0,C 180,E1 -24433.432,E2 -24433.432} C_VEL
LIN {X 0,Y 143.085,Z 377.657,A -85,B 0,C 180,E1 -24437.457,E2 -24437.457} C_VEL
LIN {X 0,Y 143.085,Z 377.661,A -85,B 0,C 180,E1 -24441.803,E2 -24441.803} C_VEL
LIN {X 0,Y 143.189,Z 377.647,A -85,B 0,C 180,E1 -24447.323,E2 -24447.323} C_VEL
LIN {X 0,Y 143.194,Z 377.646,A -85,B 0,C 180,E1 -24452.062,E2 -24452.062} C_VEL
LIN {X 0,Y 143.28,Z 377.638,A -85,B 0,C 180,E1 -24458.745,E2 -24458.745} C_VEL
LIN {X 0,Y 143.326,Z 377.626,A -85,B 0,C 180,E1 -24462.89,E2 -24462.89} C_VEL
LIN {X 0,Y 143.605,Z 377.596,A -85,B 0,C 180,E1 -24468.711,E2 -24468.711} C_VEL
LIN {X 0,Y 143.688,Z 377.58,A -85,B 0,C 180,E1 -24471.563,E2 -24471.563} C_VEL
LIN {X 0,Y 144.18,Z 377.519,A -85,B 0,C 180,E1 -24480,E2 -24480} C_VEL
LIN {X 0,Y 143.629,Z 377.588,A -85,B 0,C 180,E1 -24488.442,E2 -24488.442} C_VEL
LIN {X 0,Y 143.509,Z 377.607,A -85,B 0,C 180,E1 -24491.631,E2 -24491.631} C_VEL
LIN {X 0,Y 143.304,Z 377.627,A -85,B 0,C 180,E1 -24497.113,E2 -24497.113} C_VEL
LIN {X 0,Y 143.28,Z 377.637,A -85,B 0,C 180,E1 -24501.255,E2 -24501.255} C_VEL
LIN {X 0,Y 143.193,Z 377.646,A -85,B 0,C 180,E1 -24507.937,E2 -24507.937} C_VEL
LIN {X 0,Y 143.176,Z 377.647,A -85,B 0,C 180,E1 -24513.438,E2 -24513.438} C_VEL
LIN {X 0,Y 143.372,Z 377.627,A -85,B 0,C 180,E1 -24519.588,E2 -24519.588} C_VEL
LIN {X 0,Y 143.829,Z 377.771,A -85,B 0,C 180,E1 -24523.647,E2 -24523.647} C_VEL
LIN {X 0,Y 145.243,Z 382.997,A -85,B 0,C 180,E1 -24528.7,E2 -24528.7} C_VEL
LIN {X 0,Y 145.802,Z 385.617,A -85,B 0,C 180,E1 -24531.197,E2 -24531.197} C_VEL
LIN {X 0,Y 145.147,Z 389.017,A -85,B 0,C 180,E1 -24534.476,E2 -24534.476} C_VEL
LIN {X 0,Y 143.453,Z 396.458,A -85,B 0,C 180,E1 -24541.867,E2 -24541.867} C_VEL
LIN {X 0,Y 142.989,Z 400.374,A -85,B 0,C 180,E1 -24545.692,E2 -24545.692} C_VEL
LIN {X 0,Y 142.374,Z 413.057,A -85,B 0,C 180,E1 -24547.508,E2 -24547.508} C_VEL
LIN {X 0,Y 142.549,Z 425.734,A -85,B 0,C 180,E1 -24549.811,E2 -24549.811} C_VEL
LIN {X 0,Y 143.527,Z 439.437,A -85,B 0,C 180,E1 -24552.914,E2 -24552.914} C_VEL
LIN {X 0,Y 145.03,Z 451.516,A -85,B 0,C 180,E1 -24556.257,E2 -24556.257} C_VEL
LIN {X 0,Y 146.017,Z 457.573,A -85,B 0,C 180,E1 -24558.196,E2 -24558.196} C_VEL
LIN {X 0,Y 146.316,Z 466.363,A -85,B 0,C 180,E1 -24561.715,E2 -24561.715} C_VEL
LIN {X 0,Y 146.927,Z 474.738,A -85,B 0,C 180,E1 -24565.885,E2 -24565.885} C_VEL
LIN {X 0,Y 147.964,Z 481.382,A -85,B 0,C 180,E1 -24570,E2 -24570} C_VEL
LIN {X 0,Y 148.114,Z 483.151,A -85,B 0,C 180,E1 -24571.361,E2 -24571.361} C_VEL
LIN {X 0,Y 146.933,Z 485.499,A -85,B 0,C 180,E1 -24574.114,E2 -24574.114} C_VEL
LIN {X 0,Y 145.317,Z 488.162,A -85,B 0,C 180,E1 -24578.342,E2 -24578.342} C_VEL
LIN {X 0,Y 144.581,Z 490.637,A -85,B 0,C 180,E1 -24584.066,E2 -24584.066} C_VEL
LIN {X 0,Y 145.648,Z 492.051,A -85,B 0,C 180,E1 -24589.741,E2 -24589.741} C_VEL
LIN {X 0,Y 148.538,Z 492.544,A -85,B 0,C 180,E1 -24595.203,E2 -24595.203} C_VEL
LIN {X 0,Y 153.344,Z 492.211,A -85,B 0,C 180,E1 -24600.275,E2 -24600.275} C_VEL
LIN {X 0,Y 159.629,Z 490.99,A -85,B 0,C 180,E1 -24604.915,E2 -24604.915} C_VEL
LIN {X 0,Y 166.887,Z 488.834,A -85,B 0,C 180,E1 -24609.175,E2 -24609.175} C_VEL
LIN {X 0,Y 175.289,Z 485.819,A -85,B 0,C 180,E1 -24612.969,E2 -24612.969} C_VEL
LIN {X 0,Y 179.623,Z 484.007,A -85,B 0,C 180,E1 -24614.771,E2 -24614.771} C_VEL
LIN {X 0,Y 185.804,Z 480.975,A -85,B 0,C 180,E1 -24617.526,E2 -24617.526} C_VEL
LIN {X 0,Y 191.735,Z 477.739,A -85,B 0,C 180,E1 -24620.332,E2 -24620.332} C_VEL
LIN {X 0,Y 192.01,Z 477.302,A -85,B 0,C 180,E1 -24620.962,E2 -24620.962} C_VEL
LIN {X 0,Y 181.347,Z 478.014,A -85,B 0,C 180,E1 -24624.456,E2 -24624.456} C_VEL
LIN {X 0,Y 172.546,Z 477.382,A -85,B 0,C 180,E1 -24628.028,E2 -24628.028} C_VEL
LIN {X 0,Y 166.127,Z 475.95,A -85,B 0,C 180,E1 -24631.215,E2 -24631.215} C_VEL
LIN {X 0,Y 162.528,Z 475.065,A -85,B 0,C 180,E1 -24632.816,E2 -24632.816} C_VEL
LIN {X 0,Y 155.504,Z 473.159,A -85,B 0,C 180,E1 -24635.244,E2 -24635.244} C_VEL
LIN {X 0,Y 148.942,Z 470.566,A -85,B 0,C 180,E1 -24637.856,E2 -24637.856} C_VEL
LIN {X 0,Y 146.154,Z 468.596,A -85,B 0,C 180,E1 -24639.725,E2 -24639.725} C_VEL
LIN {X 0,Y 141.102,Z 461.997,A -85,B 0,C 180,E1 -24645.579,E2 -24645.579} C_VEL
LIN {X 0,Y 138.021,Z 454.429,A -85,B 0,C 180,E1 -24651.213,E2 -24651.213} C_VEL
LIN {X 0,Y 136.525,Z 445.221,A -85,B 0,C 180,E1 -24657.049,E2 -24657.049} C_VEL
LIN {X 0,Y 136.021,Z 436.88,A -85,B 0,C 180,E1 -24661.48,E2 -24661.48} C_VEL
LIN {X 0,Y 136.352,Z 425.265,A -85,B 0,C 180,E1 -24666.659,E2 -24666.659} C_VEL
LIN {X 0,Y 137.193,Z 414.296,A -85,B 0,C 180,E1 -24670.701,E2 -24670.701} C_VEL
LIN {X 0,Y 138.318,Z 402.304,A -85,B 0,C 180,E1 -24674.332,E2 -24674.332} C_VEL
LIN {X 0,Y 139.277,Z 392.375,A -85,B 0,C 180,E1 -24676.843,E2 -24676.843} C_VEL
LIN {X 0,Y 138.966,Z 389.571,A -85,B 0,C 180,E1 -24677.468,E2 -24677.468} C_VEL
LIN {X 0,Y 136.635,Z 378.49,A -85,B 0,C 180,E1 -24679.629,E2 -24679.629} C_VEL
LIN {X 0,Y 136.151,Z 378.523,A -85,B 0,C 180,E1 -24687.682,E2 -24687.682} C_VEL
LIN {X 0,Y 136.094,Z 378.526,A -85,B 0,C 180,E1 -24694.284,E2 -24694.284} C_VEL
LIN {X 0,Y 136.07,Z 378.535,A -85,B 0,C 180,E1 -24699.218,E2 -24699.218} C_VEL
LIN {X 0,Y 136.035,Z 378.535,A -85,B 0,C 180,E1 -24703.673,E2 -24703.673} C_VEL
LIN {X 0,Y 136.037,Z 378.539,A -85,B 0,C 180,E1 -24707.808,E2 -24707.808} C_VEL
LIN {X 0,Y 136.056,Z 378.53,A -85,B 0,C 180,E1 -24711.694,E2 -24711.694} C_VEL
LIN {X 0,Y 136.091,Z 378.532,A -85,B 0,C 180,E1 -24715.717,E2 -24715.717} C_VEL
LIN {X 0,Y 136.147,Z 378.524,A -85,B 0,C 180,E1 -24722.317,E2 -24722.317} C_VEL
LIN {X 0,Y 136.278,Z 378.504,A -85,B 0,C 180,E1 -24728.839,E2 -24728.839} C_VEL
LIN {X 0,Y 136.277,Z 378.507,A -85,B 0,C 180,E1 -24735.057,E2 -24735.057} C_VEL
LIN {X 0,Y 136.445,Z 378.483,A -85,B 0,C 180,E1 -24738.138,E2 -24738.138} C_VEL
LIN {X 0,Y 136.552,Z 378.475,A -85,B 0,C 180,E1 -24741.118,E2 -24741.118} C_VEL
LIN {X 0,Y 137.134,Z 378.404,A -85,B 0,C 180,E1 -24750,E2 -24750} C_VEL
LIN {X 0,Y 136.552,Z 378.475,A -85,B 0,C 180,E1 -24758.882,E2 -24758.882} C_VEL
LIN {X 0,Y 136.441,Z 378.484,A -85,B 0,C 180,E1 -24761.891,E2 -24761.891} C_VEL
LIN {X 0,Y 136.247,Z 378.513,A -85,B 0,C 180,E1 -24768.029,E2 -24768.029} C_VEL
LIN {X 0,Y 136.2,Z 378.514,A -85,B 0,C 180,E1 -24771.75,E2 -24771.75} C_VEL
LIN {X 0,Y 136.101,Z 378.528,A -85,B 0,C 180,E1 -24778.617,E2 -24778.617} C_VEL
LIN {X 0,Y 136.084,Z 378.533,A -85,B 0,C 180,E1 -24784.618,E2 -24784.618} C_VEL
LIN {X 0,Y 136.089,Z 378.527,A -85,B 0,C 180,E1 -24789.228,E2 -24789.228} C_VEL
LIN {X 0,Y 136.054,Z 378.537,A -85,B 0,C 180,E1 -24793.682,E2 -24793.682} C_VEL
LIN {X 0,Y 136.045,Z 378.534,A -85,B 0,C 180,E1 -24797.812,E2 -24797.812} C_VEL
LIN {X 0,Y 136.035,Z 378.539,A -85,B 0,C 180,E1 -24801.688,E2 -24801.688} C_VEL
LIN {X 0,Y 136.059,Z 378.53,A -85,B 0,C 180,E1 -24805.739,E2 -24805.739} C_VEL
LIN {X 0,Y 136.15,Z 378.524,A -85,B 0,C 180,E1 -24812.318,E2 -24812.318} C_VEL
LIN {X 0,Y 136.247,Z 378.515,A -85,B 0,C 180,E1 -24818.834,E2 -24818.834} C_VEL
LIN {X 0,Y 136.292,Z 378.507,A -85,B 0,C 180,E1 -24825.059,E2 -24825.059} C_VEL
LIN {X 0,Y 136.504,Z 378.481,A -85,B 0,C 180,E1 -24828.116,E2 -24828.116} C_VEL
LIN {X 0,Y 136.612,Z 378.461,A -85,B 0,C 180,E1 -24831.122,E2 -24831.122} C_VEL
LIN {X 0,Y 137.137,Z 378.396,A -85,B 0,C 180,E1 -24840,E2 -24840} C_VEL
LIN {X 0,Y 136.554,Z 378.47,A -85,B 0,C 180,E1 -24848.882,E2 -24848.882} C_VEL
LIN {X 0,Y 136.443,Z 378.488,A -85,B 0,C 180,E1 -24851.891,E2 -24851.891} C_VEL
LIN {X 0,Y 136.245,Z 378.508,A -85,B 0,C 180,E1 -24858.03,E2 -24858.03} C_VEL
LIN {X 0,Y 136.201,Z 378.519,A -85,B 0,C 180,E1 -24861.749,E2 -24861.749} C_VEL
LIN {X 0,Y 136.103,Z 378.531,A -85,B 0,C 180,E1 -24868.617,E2 -24868.617} C_VEL
LIN {X 0,Y 136.098,Z 378.526,A -85,B 0,C 180,E1 -24874.614,E2 -24874.614} C_VEL
LIN {X 0,Y 136.325,Z 378.504,A -85,B 0,C 180,E1 -24879.348,E2 -24879.348} C_VEL
LIN {X 0,Y 136.886,Z 378.519,A -85,B 0,C 180,E1 -24884.289,E2 -24884.289} C_VEL
LIN {X 0,Y 138.353,Z 383.782,A -85,B 0,C 180,E1 -24889.639,E2 -24889.639} C_VEL
LIN {X 0,Y 138.702,Z 385.303,A -85,B 0,C 180,E1 -24891.17,E2 -24891.17} C_VEL
LIN {X 0,Y 138.01,Z 388.63,A -85,B 0,C 180,E1 -24894.566,E2 -24894.566} C_VEL
LIN {X 0,Y 136.336,Z 395.974,A -85,B 0,C 180,E1 -24902.358,E2 -24902.358} C_VEL
LIN {X 0,Y 136.003,Z 399.117,A -85,B 0,C 180,E1 -24905.784,E2 -24905.784} C_VEL
LIN {X 0,Y 135.359,Z 412.682,A -85,B 0,C 180,E1 -24907.887,E2 -24907.887} C_VEL
LIN {X 0,Y 135.583,Z 425.254,A -85,B 0,C 180,E1 -24910.324,E2 -24910.324} C_VEL
LIN {X 0,Y 136.645,Z 438.723,A -85,B 0,C 180,E1 -24913.568,E2 -24913.568} C_VEL
LIN {X 0,Y 138.163,Z 450.182,A -85,B 0,C 180,E1 -24916.913,E2 -24916.913} C_VEL
LIN {X 0,Y 139.334,Z 456.684,A -85,B 0,C 180,E1 -24919.097,E2 -24919.097} C_VEL
LIN {X 0,Y 139.719,Z 465.308,A -85,B 0,C 180,E1 -24922.776,E2 -24922.776} C_VEL
LIN {X 0,Y 140.519,Z 473.578,A -85,B 0,C 180,E1 -24927.133,E2 -24927.133} C_VEL
LIN {X 0,Y 141.497,Z 479.266,A -85,B 0,C 180,E1 -24930.825,E2 -24930.825} C_VEL
LIN {X 0,Y 141.596,Z 480.302,A -85,B 0,C 180,E1 -24931.648,E2 -24931.648} C_VEL
LIN {X 0,Y 140.825,Z 481.965,A -85,B 0,C 180,E1 -24933.504,E2 -24933.504} C_VEL
LIN {X 0,Y 138.763,Z 485.396,A -85,B 0,C 180,E1 -24938.739,E2 -24938.739} C_VEL
LIN {X 0,Y 138.058,Z 488.112,A -85,B 0,C 180,E1 -24944.746,E2 -24944.746} C_VEL
LIN {X 0,Y 139.244,Z 489.806,A -85,B 0,C 180,E1 -24950.69,E2 -24950.69} C_VEL
LIN {X 0,Y 142.348,Z 490.574,A -85,B 0,C 180,E1 -24956.382,E2 -24956.382} C_VEL
LIN {X 0,Y 147.38,Z 490.546,A -85,B 0,C 180,E1 -24961.638,E2 -24961.638} C_VEL
LIN {X 0,Y 153.914,Z 489.663,A -85,B 0,C 180,E1 -24966.413,E2 -24966.413} C_VEL
LIN {X 0,Y 161.464,Z 487.894,A -85,B 0,C 180,E1 -24970.761,E2 -24970.761} C_VEL
